LIN {X 0,Y 411.449,Z 252.234,A -85,B 0,C 180,E1 -10446.868,E2 -10446.868} C_VEL
LIN {X 0,Y 411.346,Z 252.246,A -85,B 0,C 180,E1 -10448.846,E2 -10448.846} C_VEL
LIN {X 0,Y 411.277,Z 252.254,A -85,B 0,C 180,E1 -10451.834,E2 -10451.834} C_VEL
LIN {X 0,Y 411.252,Z 252.259,A -85,B 0,C 180,E1 -10454.854,E2 -10454.854} C_VEL
LIN {X 0,Y 411.246,Z 252.261,A -85,B 0,C 180,E1 -10457.916,E2 -10457.916} C_VEL
LIN {X 0,Y 411.19,Z 252.268,A -85,B 0,C 180,E1 -10461.035,E2 -10461.035} C_VEL
LIN {X 0,Y 411.221,Z 252.266,A -85,B 0,C 180,E1 -10464.217,E2 -10464.217} C_VEL
LIN {X 0,Y 411.206,Z 252.269,A -85,B 0,C 180,E1 -10467.483,E2 -10467.483} C_VEL
LIN {X 0,Y 411.185,Z 252.27,A -85,B 0,C 180,E1 -10470.849,E2 -10470.849} C_VEL
LIN {X 0,Y 411.202,Z 252.265,A -85,B 0,C 180,E1 -10474.335,E2 -10474.335} C_VEL
LIN {X 0,Y 411.191,Z 252.266,A -85,B 0,C 180,E1 -10477.975,E2 -10477.975} C_VEL
LIN {X 0,Y 411.179,Z 252.263,A -85,B 0,C 180,E1 -10480.506,E2 -10480.506} C_VEL
LIN {X 0,Y 411.171,Z 252.27,A -85,B 0,C 180,E1 -10483.135,E2 -10483.135} C_VEL
LIN {X 0,Y 411.163,Z 252.271,A -85,B 0,C 180,E1 -10485.883,E2 -10485.883} C_VEL
LIN {X 0,Y 411.191,Z 252.402,A -85,B 0,C 180,E1 -10487.703,E2 -10487.703} C_VEL
LIN {X 0,Y 411.989,Z 257.108,A -85,B 0,C 180,E1 -10490.865,E2 -10490.865} C_VEL
LIN {X 0,Y 412.541,Z 261.129,A -85,B 0,C 180,E1 -10493.399,E2 -10493.399} C_VEL
LIN {X 0,Y 412.54,Z 265.204,A -85,B 0,C 180,E1 -10495.794,E2 -10495.794} C_VEL
LIN {X 0,Y 412.027,Z 271.404,A -85,B 0,C 180,E1 -10499.223,E2 -10499.223} C_VEL
LIN {X 0,Y 411.468,Z 277.887,A -85,B 0,C 180,E1 -10502.646,E2 -10502.646} C_VEL
LIN {X 0,Y 411.051,Z 285.054,A -85,B 0,C 180,E1 -10506.31,E2 -10506.31} C_VEL
LIN {X 0,Y 410.714,Z 291.422,A -85,B 0,C 180,E1 -10509.465,E2 -10509.465} C_VEL
LIN {X 0,Y 410.498,Z 296.726,A -85,B 0,C 180,E1 -10512.035,E2 -10512.035} C_VEL
LIN {X 0,Y 413.257,Z 309.763,A -85,B 0,C 180,E1 -10512.581,E2 -10512.581} C_VEL
LIN {X 0,Y 415.025,Z 322.416,A -85,B 0,C 180,E1 -10513.27,E2 -10513.27} C_VEL
LIN {X 0,Y 415.335,Z 326.719,A -85,B 0,C 180,E1 -10513.535,E2 -10513.535} C_VEL
LIN {X 0,Y 414.448,Z 339.122,A -85,B 0,C 180,E1 -10514.384,E2 -10514.384} C_VEL
LIN {X 0,Y 413.537,Z 350.197,A -85,B 0,C 180,E1 -10515.355,E2 -10515.355} C_VEL
LIN {X 0,Y 412.787,Z 360.22,A -85,B 0,C 180,E1 -10516.462,E2 -10516.462} C_VEL
LIN {X 0,Y 412.105,Z 369.286,A -85,B 0,C 180,E1 -10517.692,E2 -10517.692} C_VEL
LIN {X 0,Y 411.231,Z 378.148,A -85,B 0,C 180,E1 -10519.165,E2 -10519.165} C_VEL
LIN {X 0,Y 410.716,Z 385.289,A -85,B 0,C 180,E1 -10520.645,E2 -10520.645} C_VEL
LIN {X 0,Y 410.351,Z 391.005,A -85,B 0,C 180,E1 -10522.125,E2 -10522.125} C_VEL
LIN {X 0,Y 410.045,Z 395.958,A -85,B 0,C 180,E1 -10523.776,E2 -10523.776} C_VEL
LIN {X 0,Y 410.021,Z 398.967,A -85,B 0,C 180,E1 -10525.084,E2 -10525.084} C_VEL
LIN {X 0,Y 409.925,Z 402.002,A -85,B 0,C 180,E1 -10527.052,E2 -10527.052} C_VEL
LIN {X 0,Y 409.968,Z 402.928,A -85,B 0,C 180,E1 -10528.035,E2 -10528.035} C_VEL
LIN {X 0,Y 409.937,Z 403.449,A -85,B 0,C 180,E1 -10529.018,E2 -10529.018} C_VEL
LIN {X 0,Y 409.937,Z 403.25,A -85,B 0,C 180,E1 -10530.982,E2 -10530.982} C_VEL
LIN {X 0,Y 409.968,Z 402.571,A -85,B 0,C 180,E1 -10531.965,E2 -10531.965} C_VEL
LIN {X 0,Y 409.93,Z 401.489,A -85,B 0,C 180,E1 -10532.948,E2 -10532.948} C_VEL
LIN {X 0,Y 409.933,Z 399.952,A -85,B 0,C 180,E1 -10533.932,E2 -10533.932} C_VEL
LIN {X 0,Y 410.019,Z 396.857,A -85,B 0,C 180,E1 -10535.409,E2 -10535.409} C_VEL
LIN {X 0,Y 410.168,Z 392.694,A -85,B 0,C 180,E1 -10536.889,E2 -10536.889} C_VEL
LIN {X 0,Y 410.469,Z 386.328,A -85,B 0,C 180,E1 -10538.616,E2 -10538.616} C_VEL
LIN {X 0,Y 410.875,Z 379.388,A -85,B 0,C 180,E1 -10540.097,E2 -10540.097} C_VEL
LIN {X 0,Y 411.323,Z 372.293,A -85,B 0,C 180,E1 -10541.332,E2 -10541.332} C_VEL
LIN {X 0,Y 411.945,Z 363.724,A -85,B 0,C 180,E1 -10542.563,E2 -10542.563} C_VEL
LIN {X 0,Y 412.637,Z 353.121,A -85,B 0,C 180,E1 -10543.795,E2 -10543.795} C_VEL
LIN {X 0,Y 413.317,Z 342.609,A -85,B 0,C 180,E1 -10544.777,E2 -10544.777} C_VEL
LIN {X 0,Y 414.077,Z 331.039,A -85,B 0,C 180,E1 -10545.631,E2 -10545.631} C_VEL
LIN {X 0,Y 414.293,Z 324.137,A -85,B 0,C 180,E1 -10546.043,E2 -10546.043} C_VEL
LIN {X 0,Y 412.569,Z 311.085,A -85,B 0,C 180,E1 -10546.724,E2 -10546.724} C_VEL
LIN {X 0,Y 410.476,Z 298.087,A -85,B 0,C 180,E1 -10547.21,E2 -10547.21} C_VEL
LIN {X 0,Y 410.33,Z 296.882,A -85,B 0,C 180,E1 -10547.274,E2 -10547.274} C_VEL
LIN {X 0,Y 410.588,Z 289.945,A -85,B 0,C 180,E1 -10550.542,E2 -10550.542} C_VEL
LIN {X 0,Y 410.854,Z 283.341,A -85,B 0,C 180,E1 -10553.702,E2 -10553.702} C_VEL
LIN {X 0,Y 411.165,Z 277.823,A -85,B 0,C 180,E1 -10556.385,E2 -10556.385} C_VEL
LIN {X 0,Y 411.568,Z 271.207,A -85,B 0,C 180,E1 -10559.683,E2 -10559.683} C_VEL
LIN {X 0,Y 411.984,Z 264.559,A -85,B 0,C 180,E1 -10563.084,E2 -10563.084} C_VEL
LIN {X 0,Y 412.252,Z 260.131,A -85,B 0,C 180,E1 -10565.423,E2 -10565.423} C_VEL
LIN {X 0,Y 411.793,Z 255.662,A -85,B 0,C 180,E1 -10567.908,E2 -10567.908} C_VEL
LIN {X 0,Y 411.242,Z 252.261,A -85,B 0,C 180,E1 -10569.915,E2 -10569.915} C_VEL
LIN {X 0,Y 411.159,Z 252.27,A -85,B 0,C 180,E1 -10573.134,E2 -10573.134} C_VEL
LIN {X 0,Y 411.145,Z 252.268,A -85,B 0,C 180,E1 -10575.883,E2 -10575.883} C_VEL
LIN {X 0,Y 411.155,Z 252.268,A -85,B 0,C 180,E1 -10579.492,E2 -10579.492} C_VEL
LIN {X 0,Y 411.177,Z 252.265,A -85,B 0,C 180,E1 -10582.023,E2 -10582.023} C_VEL
LIN {X 0,Y 411.197,Z 252.264,A -85,B 0,C 180,E1 -10585.122,E2 -10585.122} C_VEL
LIN {X 0,Y 411.161,Z 252.268,A -85,B 0,C 180,E1 -10588.001,E2 -10588.001} C_VEL
LIN {X 0,Y 411.174,Z 252.266,A -85,B 0,C 180,E1 -10591.406,E2 -10591.406} C_VEL
LIN {X 0,Y 411.222,Z 252.261,A -85,B 0,C 180,E1 -10594.928,E2 -10594.928} C_VEL
LIN {X 0,Y 411.199,Z 252.265,A -85,B 0,C 180,E1 -10597.912,E2 -10597.912} C_VEL
LIN {X 0,Y 411.216,Z 252.261,A -85,B 0,C 180,E1 -10601.05,E2 -10601.05} C_VEL
LIN {X 0,Y 411.247,Z 252.26,A -85,B 0,C 180,E1 -10604.13,E2 -10604.13} C_VEL
LIN {X 0,Y 411.296,Z 252.251,A -85,B 0,C 180,E1 -10607.164,E2 -10607.164} C_VEL
LIN {X 0,Y 411.285,Z 252.254,A -85,B 0,C 180,E1 -10610.16,E2 -10610.16} C_VEL
LIN {X 0,Y 411.448,Z 252.232,A -85,B 0,C 180,E1 -10613.132,E2 -10613.132} C_VEL
LIN {X 0,Y 411.302,Z 252.25,A -85,B 0,C 180,E1 -10615.098,E2 -10615.098} C_VEL
LIN {X 0,Y 411.505,Z 252.227,A -85,B 0,C 180,E1 -10618.041,E2 -10618.041} C_VEL
LIN {X 0,Y 411.635,Z 252.211,A -85,B 0,C 180,E1 -10619.999,E2 -10619.999} C_VEL
LIN {X 0,Y 411.458,Z 252.231,A -85,B 0,C 180,E1 -10622.936,E2 -10622.936} C_VEL
LIN {X 0,Y 411.452,Z 252.232,A -85,B 0,C 180,E1 -10626.866,E2 -10626.866} C_VEL
LIN {X 0,Y 411.284,Z 252.255,A -85,B 0,C 180,E1 -10629.838,E2 -10629.838} C_VEL
LIN {X 0,Y 411.295,Z 252.252,A -85,B 0,C 180,E1 -10633.103,E2 -10633.103} C_VEL
LIN {X 0,Y 411.247,Z 252.258,A -85,B 0,C 180,E1 -10636.888,E2 -10636.888} C_VEL
LIN {X 0,Y 411.22,Z 252.261,A -85,B 0,C 180,E1 -10639.986,E2 -10639.986} C_VEL
LIN {X 0,Y 411.192,Z 252.265,A -85,B 0,C 180,E1 -10643.147,E2 -10643.147} C_VEL
LIN {X 0,Y 411.227,Z 252.259,A -85,B 0,C 180,E1 -10646.38,E2 -10646.38} C_VEL
LIN {X 0,Y 411.199,Z 252.264,A -85,B 0,C 180,E1 -10649.711,E2 -10649.711} C_VEL
LIN {X 0,Y 411.195,Z 252.268,A -85,B 0,C 180,E1 -10653.155,E2 -10653.155} C_VEL
LIN {X 0,Y 411.184,Z 252.265,A -85,B 0,C 180,E1 -10656.553,E2 -10656.553} C_VEL
LIN {X 0,Y 411.217,Z 252.259,A -85,B 0,C 180,E1 -10659.73,E2 -10659.73} C_VEL
LIN {X 0,Y 411.21,Z 252.263,A -85,B 0,C 180,E1 -10663.127,E2 -10663.127} C_VEL
LIN {X 0,Y 411.164,Z 252.265,A -85,B 0,C 180,E1 -10665.879,E2 -10665.879} C_VEL
LIN {X 0,Y 411.153,Z 252.273,A -85,B 0,C 180,E1 -10668.771,E2 -10668.771} C_VEL
LIN {X 0,Y 411.188,Z 252.263,A -85,B 0,C 180,E1 -10672.027,E2 -10672.027} C_VEL
LIN {X 0,Y 411.193,Z 252.262,A -85,B 0,C 180,E1 -10675.666,E2 -10675.666} C_VEL
LIN {X 0,Y 411.177,Z 252.265,A -85,B 0,C 180,E1 -10679.152,E2 -10679.152} C_VEL
LIN {X 0,Y 411.246,Z 252.259,A -85,B 0,C 180,E1 -10682.522,E2 -10682.522} C_VEL
LIN {X 0,Y 411.155,Z 252.269,A -85,B 0,C 180,E1 -10685.781,E2 -10685.781} C_VEL
LIN {X 0,Y 411.012,Z 252.288,A -85,B 0,C 180,E1 -10687.903,E2 -10687.903} C_VEL
LIN {X 0,Y 410.972,Z 253.172,A -85,B 0,C 180,E1 -10688.954,E2 -10688.954} C_VEL
LIN {X 0,Y 410.936,Z 255.861,A -85,B 0,C 180,E1 -10691.038,E2 -10691.038} C_VEL
LIN {X 0,Y 410.798,Z 259.931,A -85,B 0,C 180,E1 -10694.114,E2 -10694.114} C_VEL
LIN {X 0,Y 410.734,Z 264.145,A -85,B 0,C 180,E1 -10697.236,E2 -10697.236} C_VEL
LIN {X 0,Y 410.55,Z 269.533,A -85,B 0,C 180,E1 -10701.138,E2 -10701.138} C_VEL
LIN {X 0,Y 410.478,Z 273.682,A -85,B 0,C 180,E1 -10704.104,E2 -10704.104} C_VEL
LIN {X 0,Y 410.463,Z 276.293,A -85,B 0,C 180,E1 -10705.858,E2 -10705.858} C_VEL
LIN {X 0,Y 412.94,Z 289.606,A -85,B 0,C 180,E1 -10706.387,E2 -10706.387} C_VEL
LIN {X 0,Y 414.786,Z 300.337,A -85,B 0,C 180,E1 -10706.965,E2 -10706.965} C_VEL
LIN {X 0,Y 414.185,Z 312.098,A -85,B 0,C 180,E1 -10707.69,E2 -10707.69} C_VEL
LIN {X 0,Y 413.496,Z 322.814,A -85,B 0,C 180,E1 -10708.539,E2 -10708.539} C_VEL
LIN {X 0,Y 412.843,Z 333.725,A -85,B 0,C 180,E1 -10709.634,E2 -10709.634} C_VEL
LIN {X 0,Y 412.126,Z 342.64,A -85,B 0,C 180,E1 -10710.733,E2 -10710.733} C_VEL
LIN {X 0,Y 411.527,Z 350.815,A -85,B 0,C 180,E1 -10711.957,E2 -10711.957} C_VEL
LIN {X 0,Y 410.964,Z 358.837,A -85,B 0,C 180,E1 -10713.431,E2 -10713.431} C_VEL
LIN {X 0,Y 410.515,Z 365.289,A -85,B 0,C 180,E1 -10714.91,E2 -10714.91} C_VEL
LIN {X 0,Y 410.331,Z 371,A -85,B 0,C 180,E1 -10716.601,E2 -10716.601} C_VEL
LIN {X 0,Y 410.063,Z 375.459,A -85,B 0,C 180,E1 -10718.376,E2 -10718.376} C_VEL
LIN {X 0,Y 409.869,Z 378.544,A -85,B 0,C 180,E1 -10720.255,E2 -10720.255} C_VEL
LIN {X 0,Y 409.188,Z 379.493,A -85,B 0,C 180,E1 -10721.067,E2 -10721.067} C_VEL
LIN {X 0,Y 406.265,Z 380.427,A -85,B 0,C 180,E1 -10722.393,E2 -10722.393} C_VEL
LIN {X 0,Y 403.808,Z 380.668,A -85,B 0,C 180,E1 -10723.468,E2 -10723.468} C_VEL
LIN {X 0,Y 402.773,Z 380.524,A -85,B 0,C 180,E1 -10724.3,E2 -10724.3} C_VEL
LIN {X 0,Y 402.701,Z 380.36,A -85,B 0,C 180,E1 -10724.582,E2 -10724.582} C_VEL
LIN {X 0,Y 402.862,Z 378.906,A -85,B 0,C 180,E1 -10726.372,E2 -10726.372} C_VEL
LIN {X 0,Y 403.081,Z 375.863,A -85,B 0,C 180,E1 -10728.29,E2 -10728.29} C_VEL
LIN {X 0,Y 403.347,Z 372.347,A -85,B 0,C 180,E1 -10729.801,E2 -10729.801} C_VEL
LIN {X 0,Y 403.78,Z 367.273,A -85,B 0,C 180,E1 -10731.439,E2 -10731.439} C_VEL
LIN {X 0,Y 404.407,Z 360.409,A -85,B 0,C 180,E1 -10733.153,E2 -10733.153} C_VEL
LIN {X 0,Y 405.074,Z 353.084,A -85,B 0,C 180,E1 -10734.607,E2 -10734.607} C_VEL
LIN {X 0,Y 405.944,Z 344.026,A -85,B 0,C 180,E1 -10736.045,E2 -10736.045} C_VEL
LIN {X 0,Y 406.753,Z 334.707,A -85,B 0,C 180,E1 -10737.249,E2 -10737.249} C_VEL
LIN {X 0,Y 407.689,Z 324.192,A -85,B 0,C 180,E1 -10738.348,E2 -10738.348} C_VEL
LIN {X 0,Y 408.433,Z 313.724,A -85,B 0,C 180,E1 -10739.225,E2 -10739.225} C_VEL
LIN {X 0,Y 409.225,Z 302.753,A -85,B 0,C 180,E1 -10739.941,E2 -10739.941} C_VEL
LIN {X 0,Y 407.639,Z 293.422,A -85,B 0,C 180,E1 -10740.531,E2 -10740.531} C_VEL
LIN {X 0,Y 404.545,Z 281.297,A -85,B 0,C 180,E1 -10741.177,E2 -10741.177} C_VEL
LIN {X 0,Y 403.264,Z 276.621,A -85,B 0,C 180,E1 -10741.397,E2 -10741.397} C_VEL
LIN {X 0,Y 403.41,Z 273.295,A -85,B 0,C 180,E1 -10743.881,E2 -10743.881} C_VEL
LIN {X 0,Y 403.581,Z 268.536,A -85,B 0,C 180,E1 -10747.552,E2 -10747.552} C_VEL
LIN {X 0,Y 403.738,Z 265.304,A -85,B 0,C 180,E1 -10750.095,E2 -10750.095} C_VEL
LIN {X 0,Y 403.957,Z 261.659,A -85,B 0,C 180,E1 -10753.056,E2 -10753.056} C_VEL
LIN {X 0,Y 404.202,Z 258.197,A -85,B 0,C 180,E1 -10755.936,E2 -10755.936} C_VEL
LIN {X 0,Y 404.237,Z 255.081,A -85,B 0,C 180,E1 -10758.652,E2 -10758.652} C_VEL
LIN {X 0,Y 404.164,Z 253.629,A -85,B 0,C 180,E1 -10759.957,E2 -10759.957} C_VEL
LIN {X 0,Y 404.135,Z 253.148,A -85,B 0,C 180,E1 -10761.494,E2 -10761.494} C_VEL
LIN {X 0,Y 404.173,Z 253.143,A -85,B 0,C 180,E1 -10764.985,E2 -10764.985} C_VEL
LIN {X 0,Y 404.133,Z 253.148,A -85,B 0,C 180,E1 -10768.555,E2 -10768.555} C_VEL
LIN {X 0,Y 404.186,Z 253.14,A -85,B 0,C 180,E1 -10772.001,E2 -10772.001} C_VEL
LIN {X 0,Y 404.166,Z 253.141,A -85,B 0,C 180,E1 -10775.335,E2 -10775.335} C_VEL
LIN {X 0,Y 404.183,Z 253.138,A -85,B 0,C 180,E1 -10778.585,E2 -10778.585} C_VEL
LIN {X 0,Y 404.203,Z 253.135,A -85,B 0,C 180,E1 -10781.763,E2 -10781.763} C_VEL
LIN {X 0,Y 404.199,Z 253.136,A -85,B 0,C 180,E1 -10784.883,E2 -10784.883} C_VEL
LIN {X 0,Y 404.246,Z 253.131,A -85,B 0,C 180,E1 -10787.96,E2 -10787.96} C_VEL
LIN {X 0,Y 404.396,Z 253.111,A -85,B 0,C 180,E1 -10792.129,E2 -10792.129} C_VEL
LIN {X 0,Y 404.409,Z 253.109,A -85,B 0,C 180,E1 -10794.016,E2 -10794.016} C_VEL
LIN {X 0,Y 404.474,Z 253.102,A -85,B 0,C 180,E1 -10798.01,E2 -10798.01} C_VEL
LIN {X 0,Y 404.598,Z 253.085,A -85,B 0,C 180,E1 -10800.001,E2 -10800.001} C_VEL
LIN {X 0,Y 404.415,Z 253.11,A -85,B 0,C 180,E1 -10802.99,E2 -10802.99} C_VEL
LIN {X 0,Y 404.401,Z 253.111,A -85,B 0,C 180,E1 -10806.989,E2 -10806.989} C_VEL
LIN {X 0,Y 404.251,Z 253.13,A -85,B 0,C 180,E1 -10810.013,E2 -10810.013} C_VEL
LIN {X 0,Y 404.26,Z 253.129,A -85,B 0,C 180,E1 -10813.213,E2 -10813.213} C_VEL
LIN {X 0,Y 404.21,Z 253.139,A -85,B 0,C 180,E1 -10817.008,E2 -10817.008} C_VEL
LIN {X 0,Y 404.158,Z 253.146,A -85,B 0,C 180,E1 -10820.353,E2 -10820.353} C_VEL
LIN {X 0,Y 404.164,Z 253.145,A -85,B 0,C 180,E1 -10823.576,E2 -10823.576} C_VEL
LIN {X 0,Y 404.168,Z 253.145,A -85,B 0,C 180,E1 -10825.769,E2 -10825.769} C_VEL
LIN {X 0,Y 404.155,Z 253.147,A -85,B 0,C 180,E1 -10829.138,E2 -10829.138} C_VEL
LIN {X 0,Y 404.137,Z 253.146,A -85,B 0,C 180,E1 -10832.623,E2 -10832.623} C_VEL
LIN {X 0,Y 404.177,Z 253.141,A -85,B 0,C 180,E1 -10835.191,E2 -10835.191} C_VEL
LIN {X 0,Y 404.152,Z 253.142,A -85,B 0,C 180,E1 -10838.758,E2 -10838.758} C_VEL
LIN {X 0,Y 404.121,Z 253.146,A -85,B 0,C 180,E1 -10841.601,E2 -10841.601} C_VEL
LIN {X 0,Y 404.144,Z 253.136,A -85,B 0,C 180,E1 -10844.523,E2 -10844.523} C_VEL
LIN {X 0,Y 404.148,Z 253.242,A -85,B 0,C 180,E1 -10847.298,E2 -10847.298} C_VEL
LIN {X 0,Y 404.833,Z 257.174,A -85,B 0,C 180,E1 -10850.035,E2 -10850.035} C_VEL
LIN {X 0,Y 405.473,Z 261.538,A -85,B 0,C 180,E1 -10852.875,E2 -10852.875} C_VEL
LIN {X 0,Y 405.591,Z 265.254,A -85,B 0,C 180,E1 -10855.124,E2 -10855.124} C_VEL
LIN {X 0,Y 405.26,Z 269.341,A -85,B 0,C 180,E1 -10857.48,E2 -10857.48} C_VEL
LIN {X 0,Y 404.841,Z 274.314,A -85,B 0,C 180,E1 -10860.228,E2 -10860.228} C_VEL
LIN {X 0,Y 404.279,Z 280.794,A -85,B 0,C 180,E1 -10863.687,E2 -10863.687} C_VEL
LIN {X 0,Y 403.902,Z 287.706,A -85,B 0,C 180,E1 -10867.254,E2 -10867.254} C_VEL
LIN {X 0,Y 403.56,Z 293.416,A -85,B 0,C 180,E1 -10870.123,E2 -10870.123} C_VEL
LIN {X 0,Y 403.447,Z 296.645,A -85,B 0,C 180,E1 -10871.655,E2 -10871.655} C_VEL
LIN {X 0,Y 406.328,Z 309.623,A -85,B 0,C 180,E1 -10872.223,E2 -10872.223} C_VEL
LIN {X 0,Y 408.108,Z 321.885,A -85,B 0,C 180,E1 -10872.909,E2 -10872.909} C_VEL
LIN {X 0,Y 408.572,Z 327.244,A -85,B 0,C 180,E1 -10873.255,E2 -10873.255} C_VEL
LIN {X 0,Y 407.646,Z 339.5,A -85,B 0,C 180,E1 -10874.116,E2 -10874.116} C_VEL
LIN {X 0,Y 406.684,Z 350.557,A -85,B 0,C 180,E1 -10875.113,E2 -10875.113} C_VEL
LIN {X 0,Y 405.889,Z 360.376,A -85,B 0,C 180,E1 -10876.227,E2 -10876.227} C_VEL
LIN {X 0,Y 405.16,Z 369.383,A -85,B 0,C 180,E1 -10877.478,E2 -10877.478} C_VEL
LIN {X 0,Y 404.228,Z 378.195,A -85,B 0,C 180,E1 -10878.975,E2 -10878.975} C_VEL
LIN {X 0,Y 403.684,Z 385.28,A -85,B 0,C 180,E1 -10880.48,E2 -10880.48} C_VEL
LIN {X 0,Y 403.296,Z 390.949,A -85,B 0,C 180,E1 -10881.986,E2 -10881.986} C_VEL
LIN {X 0,Y 402.942,Z 396.246,A -85,B 0,C 180,E1 -10883.82,E2 -10883.82} C_VEL
LIN {X 0,Y 402.933,Z 398.844,A -85,B 0,C 180,E1 -10884.997,E2 -10884.997} C_VEL
LIN {X 0,Y 402.824,Z 401.848,A -85,B 0,C 180,E1 -10887,E2 -10887} C_VEL
LIN {X 0,Y 402.866,Z 402.76,A -85,B 0,C 180,E1 -10888.001,E2 -10888.001} C_VEL
LIN {X 0,Y 402.864,Z 403.257,A -85,B 0,C 180,E1 -10889,E2 -10889} C_VEL
LIN {X 0,Y 402.864,Z 403.031,A -85,B 0,C 180,E1 -10891,E2 -10891} C_VEL
LIN {X 0,Y 402.881,Z 402.339,A -85,B 0,C 180,E1 -10891.999,E2 -10891.999} C_VEL
LIN {X 0,Y 402.829,Z 401.232,A -85,B 0,C 180,E1 -10893,E2 -10893} C_VEL
LIN {X 0,Y 402.854,Z 399.679,A -85,B 0,C 180,E1 -10894.001,E2 -10894.001} C_VEL
LIN {X 0,Y 402.917,Z 396.553,A -85,B 0,C 180,E1 -10895.505,E2 -10895.505} C_VEL
LIN {X 0,Y 403.08,Z 392.356,A -85,B 0,C 180,E1 -10897.01,E2 -10897.01} C_VEL
LIN {X 0,Y 403.406,Z 385.953,A -85,B 0,C 180,E1 -10898.768,E2 -10898.768} C_VEL
LIN {X 0,Y 403.816,Z 378.963,A -85,B 0,C 180,E1 -10900.276,E2 -10900.276} C_VEL
LIN {X 0,Y 404.447,Z 370.19,A -85,B 0,C 180,E1 -10901.781,E2 -10901.781} C_VEL
LIN {X 0,Y 405.07,Z 361.192,A -85,B 0,C 180,E1 -10903.035,E2 -10903.035} C_VEL
LIN {X 0,Y 405.756,Z 351.295,A -85,B 0,C 180,E1 -10904.161,E2 -10904.161} C_VEL
LIN {X 0,Y 406.523,Z 340.37,A -85,B 0,C 180,E1 -10905.158,E2 -10905.158} C_VEL
LIN {X 0,Y 407.314,Z 328.101,A -85,B 0,C 180,E1 -10906.026,E2 -10906.026} C_VEL
LIN {X 0,Y 407.049,Z 322.118,A -85,B 0,C 180,E1 -10906.388,E2 -10906.388} C_VEL
LIN {X 0,Y 405.243,Z 309.092,A -85,B 0,C 180,E1 -10907.056,E2 -10907.056} C_VEL
LIN {X 0,Y 403.259,Z 296.712,A -85,B 0,C 180,E1 -10907.528,E2 -10907.528} C_VEL
LIN {X 0,Y 403.549,Z 289.665,A -85,B 0,C 180,E1 -10910.917,E2 -10910.917} C_VEL
LIN {X 0,Y 403.853,Z 283.072,A -85,B 0,C 180,E1 -10914.139,E2 -10914.139} C_VEL
LIN {X 0,Y 404.131,Z 277.567,A -85,B 0,C 180,E1 -10916.881,E2 -10916.881} C_VEL
LIN {X 0,Y 404.59,Z 270.943,A -85,B 0,C 180,E1 -10920.248,E2 -10920.248} C_VEL
LIN {X 0,Y 405.02,Z 264.295,A -85,B 0,C 180,E1 -10923.729,E2 -10923.729} C_VEL
LIN {X 0,Y 405.16,Z 259.864,A -85,B 0,C 180,E1 -10926.14,E2 -10926.14} C_VEL
LIN {X 0,Y 404.568,Z 255.407,A -85,B 0,C 180,E1 -10928.709,E2 -10928.709} C_VEL
LIN {X 0,Y 404.199,Z 253.139,A -85,B 0,C 180,E1 -10930.088,E2 -10930.088} C_VEL
LIN {X 0,Y 404.116,Z 253.144,A -85,B 0,C 180,E1 -10934.077,E2 -10934.077} C_VEL
LIN {X 0,Y 404.073,Z 253.151,A -85,B 0,C 180,E1 -10937.286,E2 -10937.286} C_VEL
LIN {X 0,Y 404.13,Z 253.142,A -85,B 0,C 180,E1 -10939.95,E2 -10939.95} C_VEL
LIN {X 0,Y 404.127,Z 253.145,A -85,B 0,C 180,E1 -10943.125,E2 -10943.125} C_VEL
LIN {X 0,Y 404.134,Z 253.144,A -85,B 0,C 180,E1 -10946.186,E2 -10946.186} C_VEL
LIN {X 0,Y 404.14,Z 253.142,A -85,B 0,C 180,E1 -10949.713,E2 -10949.713} C_VEL
LIN {X 0,Y 404.119,Z 253.146,A -85,B 0,C 180,E1 -10953.116,E2 -10953.116} C_VEL
LIN {X 0,Y 404.152,Z 253.143,A -85,B 0,C 180,E1 -10956.423,E2 -10956.423} C_VEL
LIN {X 0,Y 404.186,Z 253.138,A -85,B 0,C 180,E1 -10959.873,E2 -10959.873} C_VEL
LIN {X 0,Y 404.21,Z 253.134,A -85,B 0,C 180,E1 -10962.992,E2 -10962.992} C_VEL
LIN {X 0,Y 404.276,Z 253.126,A -85,B 0,C 180,E1 -10966.938,E2 -10966.938} C_VEL
LIN {X 0,Y 404.251,Z 253.131,A -85,B 0,C 180,E1 -10969.987,E2 -10969.987} C_VEL
LIN {X 0,Y 404.395,Z 253.11,A -85,B 0,C 180,E1 -10973.011,E2 -10973.011} C_VEL
LIN {X 0,Y 404.274,Z 253.126,A -85,B 0,C 180,E1 -10975.012,E2 -10975.012} C_VEL
LIN {X 0,Y 404.474,Z 253.103,A -85,B 0,C 180,E1 -10978.007,E2 -10978.007} C_VEL
LIN {X 0,Y 404.604,Z 253.087,A -85,B 0,C 180,E1 -10979.999,E2 -10979.999} C_VEL
LIN {X 0,Y 404.415,Z 253.108,A -85,B 0,C 180,E1 -10982.987,E2 -10982.987} C_VEL
LIN {X 0,Y 404.403,Z 253.11,A -85,B 0,C 180,E1 -10986.986,E2 -10986.986} C_VEL
LIN {X 0,Y 404.25,Z 253.131,A -85,B 0,C 180,E1 -10990.011,E2 -10990.011} C_VEL
LIN {X 0,Y 404.256,Z 253.129,A -85,B 0,C 180,E1 -10993.21,E2 -10993.21} C_VEL
LIN {X 0,Y 404.205,Z 253.135,A -85,B 0,C 180,E1 -10997.006,E2 -10997.006} C_VEL
LIN {X 0,Y 404.153,Z 253.14,A -85,B 0,C 180,E1 -11000.351,E2 -11000.351} C_VEL
LIN {X 0,Y 404.158,Z 253.143,A -85,B 0,C 180,E1 -11003.574,E2 -11003.574} C_VEL
LIN {X 0,Y 404.172,Z 253.139,A -85,B 0,C 180,E1 -11005.766,E2 -11005.766} C_VEL
LIN {X 0,Y 404.186,Z 253.136,A -85,B 0,C 180,E1 -11007.999,E2 -11007.999} C_VEL
LIN {X 0,Y 404.131,Z 253.145,A -85,B 0,C 180,E1 -11011.558,E2 -11011.558} C_VEL
LIN {X 0,Y 404.174,Z 253.141,A -85,B 0,C 180,E1 -11015.015,E2 -11015.015} C_VEL
LIN {X 0,Y 404.152,Z 253.142,A -85,B 0,C 180,E1 -11018.755,E2 -11018.755} C_VEL
LIN {X 0,Y 404.179,Z 253.136,A -85,B 0,C 180,E1 -11021.61,E2 -11021.61} C_VEL
LIN {X 0,Y 404.178,Z 253.138,A -85,B 0,C 180,E1 -11024.528,E2 -11024.528} C_VEL
LIN {X 0,Y 404.127,Z 253.143,A -85,B 0,C 180,E1 -11027.296,E2 -11027.296} C_VEL
LIN {X 0,Y 404.157,Z 253.138,A -85,B 0,C 180,E1 -11029.955,E2 -11029.955} C_VEL
LIN {X 0,Y 404.127,Z 253.144,A -85,B 0,C 180,E1 -11033.124,E2 -11033.124} C_VEL
LIN {X 0,Y 404.133,Z 253.144,A -85,B 0,C 180,E1 -11036.187,E2 -11036.187} C_VEL
LIN {X 0,Y 404.133,Z 253.142,A -85,B 0,C 180,E1 -11039.715,E2 -11039.715} C_VEL
LIN {X 0,Y 404.18,Z 253.137,A -85,B 0,C 180,E1 -11043.122,E2 -11043.122} C_VEL
LIN {X 0,Y 404.07,Z 253.153,A -85,B 0,C 180,E1 -11046.42,E2 -11046.42} C_VEL
LIN {X 0,Y 404.033,Z 253.155,A -85,B 0,C 180,E1 -11047.501,E2 -11047.501} C_VEL
LIN {X 0,Y 403.911,Z 253.541,A -85,B 0,C 180,E1 -11048.568,E2 -11048.568} C_VEL
LIN {X 0,Y 403.921,Z 256.251,A -85,B 0,C 180,E1 -11050.696,E2 -11050.696} C_VEL
LIN {X 0,Y 403.777,Z 260.321,A -85,B 0,C 180,E1 -11053.83,E2 -11053.83} C_VEL
LIN {X 0,Y 403.678,Z 264.724,A -85,B 0,C 180,E1 -11057.142,E2 -11057.142} C_VEL
LIN {X 0,Y 403.471,Z 269.943,A -85,B 0,C 180,E1 -11060.981,E2 -11060.981} C_VEL
LIN {X 0,Y 403.426,Z 274.141,A -85,B 0,C 180,E1 -11064,E2 -11064} C_VEL
LIN {X 0,Y 403.422,Z 276.478,A -85,B 0,C 180,E1 -11065.598,E2 -11065.598} C_VEL
LIN {X 0,Y 405.857,Z 289.453,A -85,B 0,C 180,E1 -11066.121,E2 -11066.121} C_VEL
LIN {X 0,Y 407.861,Z 300.461,A -85,B 0,C 180,E1 -11066.728,E2 -11066.728} C_VEL
LIN {X 0,Y 407.228,Z 313.099,A -85,B 0,C 180,E1 -11067.527,E2 -11067.527} C_VEL
LIN {X 0,Y 406.453,Z 324.935,A -85,B 0,C 180,E1 -11068.514,E2 -11068.514} C_VEL
LIN {X 0,Y 405.74,Z 335.48,A -85,B 0,C 180,E1 -11069.628,E2 -11069.628} C_VEL
LIN {X 0,Y 405.054,Z 344.128,A -85,B 0,C 180,E1 -11070.746,E2 -11070.746} C_VEL
LIN {X 0,Y 404.417,Z 352.096,A -85,B 0,C 180,E1 -11071.992,E2 -11071.992} C_VEL
LIN {X 0,Y 403.884,Z 359.905,A -85,B 0,C 180,E1 -11073.492,E2 -11073.492} C_VEL
LIN {X 0,Y 403.42,Z 366.158,A -85,B 0,C 180,E1 -11074.997,E2 -11074.997} C_VEL
LIN {X 0,Y 403.243,Z 371.346,A -85,B 0,C 180,E1 -11076.584,E2 -11076.584} C_VEL
LIN {X 0,Y 403.029,Z 374.978,A -85,B 0,C 180,E1 -11078.019,E2 -11078.019} C_VEL
LIN {X 0,Y 402.861,Z 376.972,A -85,B 0,C 180,E1 -11079.033,E2 -11079.033} C_VEL
LIN {X 0,Y 402.772,Z 378.764,A -85,B 0,C 180,E1 -11080.246,E2 -11080.246} C_VEL
LIN {X 0,Y 402.801,Z 380.368,A -85,B 0,C 180,E1 -11082.085,E2 -11082.085} C_VEL
LIN {X 0,Y 402.701,Z 380.682,A -85,B 0,C 180,E1 -11083.113,E2 -11083.113} C_VEL
LIN {X 0,Y 402.701,Z 380.36,A -85,B 0,C 180,E1 -11084.582,E2 -11084.582} C_VEL
LIN {X 0,Y 402.082,Z 379.899,A -85,B 0,C 180,E1 -11085.414,E2 -11085.414} C_VEL
LIN {X 0,Y 399.332,Z 378.588,A -85,B 0,C 180,E1 -11086.764,E2 -11086.764} C_VEL
LIN {X 0,Y 397.047,Z 377.068,A -85,B 0,C 180,E1 -11087.842,E2 -11087.842} C_VEL
LIN {X 0,Y 396.141,Z 375.586,A -85,B 0,C 180,E1 -11088.662,E2 -11088.662} C_VEL
LIN {X 0,Y 396.109,Z 375.007,A -85,B 0,C 180,E1 -11088.937,E2 -11088.937} C_VEL
LIN {X 0,Y 396.521,Z 370.309,A -85,B 0,C 180,E1 -11090.761,E2 -11090.761} C_VEL
LIN {X 0,Y 397.126,Z 363.752,A -85,B 0,C 180,E1 -11092.638,E2 -11092.638} C_VEL
LIN {X 0,Y 397.812,Z 356.506,A -85,B 0,C 180,E1 -11094.251,E2 -11094.251} C_VEL
LIN {X 0,Y 398.693,Z 348.09,A -85,B 0,C 180,E1 -11095.737,E2 -11095.737} C_VEL
LIN {X 0,Y 399.589,Z 338.796,A -85,B 0,C 180,E1 -11097.07,E2 -11097.07} C_VEL
LIN {X 0,Y 400.574,Z 328.368,A -85,B 0,C 180,E1 -11098.275,E2 -11098.275} C_VEL
LIN {X 0,Y 401.527,Z 316.589,A -85,B 0,C 180,E1 -11099.346,E2 -11099.346} C_VEL
LIN {X 0,Y 402.454,Z 304.784,A -85,B 0,C 180,E1 -11100.174,E2 -11100.174} C_VEL
LIN {X 0,Y 401.863,Z 299.29,A -85,B 0,C 180,E1 -11100.539,E2 -11100.539} C_VEL
LIN {X 0,Y 399.046,Z 286.807,A -85,B 0,C 180,E1 -11101.291,E2 -11101.291} C_VEL
LIN {X 0,Y 396.217,Z 276.808,A -85,B 0,C 180,E1 -11101.809,E2 -11101.809} C_VEL
LIN {X 0,Y 396.381,Z 273.194,A -85,B 0,C 180,E1 -11104.566,E2 -11104.566} C_VEL
LIN {X 0,Y 396.6,Z 268.402,A -85,B 0,C 180,E1 -11108.331,E2 -11108.331} C_VEL
LIN {X 0,Y 396.812,Z 263.973,A -85,B 0,C 180,E1 -11111.94,E2 -11111.94} C_VEL
LIN {X 0,Y 397.09,Z 260.236,A -85,B 0,C 180,E1 -11115.067,E2 -11115.067} C_VEL
LIN {X 0,Y 397.235,Z 256.878,A -85,B 0,C 180,E1 -11117.993,E2 -11117.993} C_VEL
LIN {X 0,Y 397.086,Z 254.22,A -85,B 0,C 180,E1 -11120.422,E2 -11120.422} C_VEL
LIN {X 0,Y 397.088,Z 254.023,A -85,B 0,C 180,E1 -11123.006,E2 -11123.006} C_VEL
LIN {X 0,Y 397.106,Z 254.024,A -85,B 0,C 180,E1 -11126.283,E2 -11126.283} C_VEL
LIN {X 0,Y 397.102,Z 254.023,A -85,B 0,C 180,E1 -11130.134,E2 -11130.134} C_VEL
LIN {X 0,Y 397.183,Z 254.01,A -85,B 0,C 180,E1 -11132.611,E2 -11132.611} C_VEL
LIN {X 0,Y 397.123,Z 254.019,A -85,B 0,C 180,E1 -11135.983,E2 -11135.983} C_VEL
LIN {X 0,Y 397.144,Z 254.015,A -85,B 0,C 180,E1 -11139.274,E2 -11139.274} C_VEL
LIN {X 0,Y 397.173,Z 254.011,A -85,B 0,C 180,E1 -11142.845,E2 -11142.845} C_VEL
LIN {X 0,Y 397.167,Z 254.01,A -85,B 0,C 180,E1 -11145.658,E2 -11145.658} C_VEL
LIN {X 0,Y 397.189,Z 254.011,A -85,B 0,C 180,E1 -11148.778,E2 -11148.778} C_VEL
LIN {X 0,Y 397.352,Z 253.989,A -85,B 0,C 180,E1 -11152.076,E2 -11152.076} C_VEL
LIN {X 0,Y 397.244,Z 254.003,A -85,B 0,C 180,E1 -11154.926,E2 -11154.926} C_VEL
LIN {X 0,Y 397.443,Z 253.978,A -85,B 0,C 180,E1 -11157.974,E2 -11157.974} C_VEL
LIN {X 0,Y 397.568,Z 253.961,A -85,B 0,C 180,E1 -11160.001,E2 -11160.001} C_VEL
LIN {X 0,Y 397.373,Z 253.987,A -85,B 0,C 180,E1 -11163.043,E2 -11163.043} C_VEL
LIN {X 0,Y 397.354,Z 253.989,A -85,B 0,C 180,E1 -11167.113,E2 -11167.113} C_VEL
LIN {X 0,Y 397.211,Z 254.007,A -85,B 0,C 180,E1 -11170.192,E2 -11170.192} C_VEL
LIN {X 0,Y 397.22,Z 254.005,A -85,B 0,C 180,E1 -11173.322,E2 -11173.322} C_VEL
LIN {X 0,Y 397.176,Z 254.015,A -85,B 0,C 180,E1 -11177.156,E2 -11177.156} C_VEL
LIN {X 0,Y 397.097,Z 254.023,A -85,B 0,C 180,E1 -11180.731,E2 -11180.731} C_VEL
LIN {X 0,Y 397.127,Z 254.021,A -85,B 0,C 180,E1 -11184.02,E2 -11184.02} C_VEL
LIN {X 0,Y 397.136,Z 254.022,A -85,B 0,C 180,E1 -11187.396,E2 -11187.396} C_VEL
LIN {X 0,Y 397.074,Z 254.028,A -85,B 0,C 180,E1 -11190.884,E2 -11190.884} C_VEL
LIN {X 0,Y 397.122,Z 254.019,A -85,B 0,C 180,E1 -11194.495,E2 -11194.495} C_VEL
LIN {X 0,Y 397.1,Z 254.023,A -85,B 0,C 180,E1 -11198.276,E2 -11198.276} C_VEL
LIN {X 0,Y 397.087,Z 254.02,A -85,B 0,C 180,E1 -11200.91,E2 -11200.91} C_VEL
LIN {X 0,Y 397.1,Z 254.022,A -85,B 0,C 180,E1 -11203.65,E2 -11203.65} C_VEL
LIN {X 0,Y 397.1,Z 254.074,A -85,B 0,C 180,E1 -11206.876,E2 -11206.876} C_VEL
LIN {X 0,Y 397.713,Z 257.682,A -85,B 0,C 180,E1 -11209.453,E2 -11209.453} C_VEL
LIN {X 0,Y 398.425,Z 262.288,A -85,B 0,C 180,E1 -11212.541,E2 -11212.541} C_VEL
LIN {X 0,Y 398.587,Z 266.299,A -85,B 0,C 180,E1 -11215.038,E2 -11215.038} C_VEL
LIN {X 0,Y 398.152,Z 271.416,A -85,B 0,C 180,E1 -11218.026,E2 -11218.026} C_VEL
LIN {X 0,Y 397.67,Z 276.605,A -85,B 0,C 180,E1 -11220.922,E2 -11220.922} C_VEL
LIN {X 0,Y 397.111,Z 283.913,A -85,B 0,C 180,E1 -11224.866,E2 -11224.866} C_VEL
LIN {X 0,Y 396.733,Z 290.229,A -85,B 0,C 180,E1 -11228.161,E2 -11228.161} C_VEL
LIN {X 0,Y 396.398,Z 296.384,A -85,B 0,C 180,E1 -11231.256,E2 -11231.256} C_VEL
LIN {X 0,Y 399.45,Z 309.853,A -85,B 0,C 180,E1 -11231.868,E2 -11231.868} C_VEL
LIN {X 0,Y 401.299,Z 322.142,A -85,B 0,C 180,E1 -11232.581,E2 -11232.581} C_VEL
LIN {X 0,Y 401.698,Z 329.828,A -85,B 0,C 180,E1 -11233.091,E2 -11233.091} C_VEL
LIN {X 0,Y 400.716,Z 341.427,A -85,B 0,C 180,E1 -11233.965,E2 -11233.965} C_VEL
LIN {X 0,Y 399.611,Z 353.087,A -85,B 0,C 180,E1 -11235.096,E2 -11235.096} C_VEL
LIN {X 0,Y 398.839,Z 362.493,A -85,B 0,C 180,E1 -11236.239,E2 -11236.239} C_VEL
LIN {X 0,Y 398.066,Z 371.109,A -85,B 0,C 180,E1 -11237.51,E2 -11237.51} C_VEL
LIN {X 0,Y 397.145,Z 379.501,A -85,B 0,C 180,E1 -11239.034,E2 -11239.034} C_VEL
LIN {X 0,Y 396.576,Z 386.274,A -85,B 0,C 180,E1 -11240.565,E2 -11240.565} C_VEL
LIN {X 0,Y 396.154,Z 392.514,A -85,B 0,C 180,E1 -11242.354,E2 -11242.354} C_VEL
LIN {X 0,Y 395.831,Z 397.271,A -85,B 0,C 180,E1 -11244.194,E2 -11244.194} C_VEL
LIN {X 0,Y 395.776,Z 400.411,A -85,B 0,C 180,E1 -11245.927,E2 -11245.927} C_VEL
LIN {X 0,Y 395.763,Z 402.596,A -85,B 0,C 180,E1 -11247.965,E2 -11247.965} C_VEL
LIN {X 0,Y 395.792,Z 403.065,A -85,B 0,C 180,E1 -11248.983,E2 -11248.983} C_VEL
LIN {X 0,Y 395.793,Z 402.809,A -85,B 0,C 180,E1 -11251.017,E2 -11251.017} C_VEL
LIN {X 0,Y 395.779,Z 402.102,A -85,B 0,C 180,E1 -11252.035,E2 -11252.035} C_VEL
LIN {X 0,Y 395.732,Z 400.964,A -85,B 0,C 180,E1 -11253.054,E2 -11253.054} C_VEL
LIN {X 0,Y 395.777,Z 399.396,A -85,B 0,C 180,E1 -11254.073,E2 -11254.073} C_VEL
LIN {X 0,Y 395.829,Z 395.746,A -85,B 0,C 180,E1 -11255.804,E2 -11255.804} C_VEL
LIN {X 0,Y 396.068,Z 390.362,A -85,B 0,C 180,E1 -11257.648,E2 -11257.648} C_VEL
LIN {X 0,Y 396.477,Z 383.367,A -85,B 0,C 180,E1 -11259.437,E2 -11259.437} C_VEL
LIN {X 0,Y 396.964,Z 375.786,A -85,B 0,C 180,E1 -11260.971,E2 -11260.971} C_VEL
LIN {X 0,Y 397.627,Z 368.046,A -85,B 0,C 180,E1 -11262.245,E2 -11262.245} C_VEL
LIN {X 0,Y 398.279,Z 359.07,A -85,B 0,C 180,E1 -11263.463,E2 -11263.463} C_VEL
LIN {X 0,Y 398.999,Z 348.074,A -85,B 0,C 180,E1 -11264.667,E2 -11264.667} C_VEL
LIN {X 0,Y 399.847,Z 336.393,A -85,B 0,C 180,E1 -11265.678,E2 -11265.678} C_VEL
LIN {X 0,Y 400.436,Z 325.959,A -85,B 0,C 180,E1 -11266.386,E2 -11266.386} C_VEL
LIN {X 0,Y 398.763,Z 312.947,A -85,B 0,C 180,E1 -11267.124,E2 -11267.124} C_VEL
LIN {X 0,Y 396.635,Z 299.439,A -85,B 0,C 180,E1 -11267.679,E2 -11267.679} C_VEL
LIN {X 0,Y 396.19,Z 296.549,A -85,B 0,C 180,E1 -11267.784,E2 -11267.784} C_VEL
LIN {X 0,Y 396.526,Z 289.37,A -85,B 0,C 180,E1 -11271.305,E2 -11271.305} C_VEL
LIN {X 0,Y 396.892,Z 281.692,A -85,B 0,C 180,E1 -11275.149,E2 -11275.149} C_VEL
LIN {X 0,Y 397.291,Z 275.075,A -85,B 0,C 180,E1 -11278.53,E2 -11278.53} C_VEL
LIN {X 0,Y 397.682,Z 269.583,A -85,B 0,C 180,E1 -11281.414,E2 -11281.414} C_VEL
LIN {X 0,Y 398.173,Z 262.927,A -85,B 0,C 180,E1 -11285.004,E2 -11285.004} C_VEL
LIN {X 0,Y 397.921,Z 258.793,A -85,B 0,C 180,E1 -11287.364,E2 -11287.364} C_VEL
LIN {X 0,Y 397.152,Z 254.017,A -85,B 0,C 180,E1 -11290.227,E2 -11290.227} C_VEL
LIN {X 0,Y 397.084,Z 254.02,A -85,B 0,C 180,E1 -11293.65,E2 -11293.65} C_VEL
LIN {X 0,Y 397.033,Z 254.029,A -85,B 0,C 180,E1 -11296.53,E2 -11296.53} C_VEL
LIN {X 0,Y 397.083,Z 254.023,A -85,B 0,C 180,E1 -11300.418,E2 -11300.418} C_VEL
LIN {X 0,Y 397.089,Z 254.022,A -85,B 0,C 180,E1 -11303.003,E2 -11303.003} C_VEL
LIN {X 0,Y 397.108,Z 254.021,A -85,B 0,C 180,E1 -11306.725,E2 -11306.725} C_VEL
LIN {X 0,Y 397.113,Z 254.02,A -85,B 0,C 180,E1 -11310.294,E2 -11310.294} C_VEL
LIN {X 0,Y 397.083,Z 254.021,A -85,B 0,C 180,E1 -11313.737,E2 -11313.737} C_VEL
LIN {X 0,Y 397.098,Z 254.02,A -85,B 0,C 180,E1 -11317.084,E2 -11317.084} C_VEL
LIN {X 0,Y 397.142,Z 254.017,A -85,B 0,C 180,E1 -11320.351,E2 -11320.351} C_VEL
LIN {X 0,Y 397.16,Z 254.012,A -85,B 0,C 180,E1 -11323.552,E2 -11323.552} C_VEL
LIN {X 0,Y 397.223,Z 254.005,A -85,B 0,C 180,E1 -11326.701,E2 -11326.701} C_VEL
LIN {X 0,Y 397.21,Z 254.008,A -85,B 0,C 180,E1 -11329.808,E2 -11329.808} C_VEL
LIN {X 0,Y 397.345,Z 253.989,A -85,B 0,C 180,E1 -11332.887,E2 -11332.887} C_VEL
LIN {X 0,Y 397.246,Z 254.001,A -85,B 0,C 180,E1 -11334.924,E2 -11334.924} C_VEL
LIN {X 0,Y 397.443,Z 253.979,A -85,B 0,C 180,E1 -11337.972,E2 -11337.972} C_VEL
LIN {X 0,Y 397.574,Z 253.963,A -85,B 0,C 180,E1 -11339.999,E2 -11339.999} C_VEL
LIN {X 0,Y 397.374,Z 253.985,A -85,B 0,C 180,E1 -11343.04,E2 -11343.04} C_VEL
LIN {X 0,Y 397.355,Z 253.988,A -85,B 0,C 180,E1 -11347.111,E2 -11347.111} C_VEL
LIN {X 0,Y 397.209,Z 254.007,A -85,B 0,C 180,E1 -11350.19,E2 -11350.19} C_VEL
LIN {X 0,Y 397.217,Z 254.006,A -85,B 0,C 180,E1 -11353.32,E2 -11353.32} C_VEL
LIN {X 0,Y 397.171,Z 254.012,A -85,B 0,C 180,E1 -11357.154,E2 -11357.154} C_VEL
LIN {X 0,Y 397.092,Z 254.02,A -85,B 0,C 180,E1 -11360.729,E2 -11360.729} C_VEL
LIN {X 0,Y 397.122,Z 254.016,A -85,B 0,C 180,E1 -11364.017,E2 -11364.017} C_VEL
LIN {X 0,Y 397.183,Z 254.013,A -85,B 0,C 180,E1 -11367.389,E2 -11367.389} C_VEL
LIN {X 0,Y 397.073,Z 254.024,A -85,B 0,C 180,E1 -11370.881,E2 -11370.881} C_VEL
LIN {X 0,Y 397.114,Z 254.017,A -85,B 0,C 180,E1 -11374.493,E2 -11374.493} C_VEL
LIN {X 0,Y 397.098,Z 254.018,A -85,B 0,C 180,E1 -11378.274,E2 -11378.274} C_VEL
LIN {X 0,Y 397.144,Z 254.012,A -85,B 0,C 180,E1 -11381.993,E2 -11381.993} C_VEL
LIN {X 0,Y 397.101,Z 254.021,A -85,B 0,C 180,E1 -11385.064,E2 -11385.064} C_VEL
LIN {X 0,Y 397.055,Z 254.023,A -85,B 0,C 180,E1 -11388.02,E2 -11388.02} C_VEL
LIN {X 0,Y 397.12,Z 254.017,A -85,B 0,C 180,E1 -11391.138,E2 -11391.138} C_VEL
LIN {X 0,Y 397.108,Z 254.022,A -85,B 0,C 180,E1 -11394.496,E2 -11394.496} C_VEL
LIN {X 0,Y 397.066,Z 254.023,A -85,B 0,C 180,E1 -11397.928,E2 -11397.928} C_VEL
LIN {X 0,Y 397.109,Z 254.017,A -85,B 0,C 180,E1 -11401.456,E2 -11401.456} C_VEL
LIN {X 0,Y 397.112,Z 254.017,A -85,B 0,C 180,E1 -11403.741,E2 -11403.741} C_VEL
LIN {X 0,Y 396.993,Z 254.032,A -85,B 0,C 180,E1 -11407.079,E2 -11407.079} C_VEL
LIN {X 0,Y 396.87,Z 254.052,A -85,B 0,C 180,E1 -11408.169,E2 -11408.169} C_VEL
LIN {X 0,Y 396.881,Z 256.615,A -85,B 0,C 180,E1 -11410.34,E2 -11410.34} C_VEL
LIN {X 0,Y 396.742,Z 260.717,A -85,B 0,C 180,E1 -11413.535,E2 -11413.535} C_VEL
LIN {X 0,Y 396.612,Z 265.321,A -85,B 0,C 180,E1 -11417.052,E2 -11417.052} C_VEL
LIN {X 0,Y 396.411,Z 270.377,A -85,B 0,C 180,E1 -11420.819,E2 -11420.819} C_VEL
LIN {X 0,Y 396.377,Z 274.563,A -85,B 0,C 180,E1 -11423.893,E2 -11423.893} C_VEL
LIN {X 0,Y 396.337,Z 276.543,A -85,B 0,C 180,E1 -11425.328,E2 -11425.328} C_VEL
LIN {X 0,Y 398.867,Z 289.892,A -85,B 0,C 180,E1 -11425.879,E2 -11425.879} C_VEL
LIN {X 0,Y 400.958,Z 301.653,A -85,B 0,C 180,E1 -11426.546,E2 -11426.546} C_VEL
LIN {X 0,Y 400.267,Z 314.081,A -85,B 0,C 180,E1 -11427.358,E2 -11427.358} C_VEL
LIN {X 0,Y 399.486,Z 325.717,A -85,B 0,C 180,E1 -11428.362,E2 -11428.362} C_VEL
LIN {X 0,Y 398.739,Z 336.166,A -85,B 0,C 180,E1 -11429.495,E2 -11429.495} C_VEL
LIN {X 0,Y 397.979,Z 345.611,A -85,B 0,C 180,E1 -11430.759,E2 -11430.759} C_VEL
LIN {X 0,Y 397.198,Z 354.711,A -85,B 0,C 180,E1 -11432.282,E2 -11432.282} C_VEL
LIN {X 0,Y 396.71,Z 362.033,A -85,B 0,C 180,E1 -11433.809,E2 -11433.809} C_VEL
LIN {X 0,Y 396.331,Z 367.016,A -85,B 0,C 180,E1 -11435.087,E2 -11435.087} C_VEL
LIN {X 0,Y 396.16,Z 371.708,A -85,B 0,C 180,E1 -11436.574,E2 -11436.574} C_VEL
LIN {X 0,Y 395.903,Z 375.571,A -85,B 0,C 180,E1 -11438.164,E2 -11438.164} C_VEL
LIN {X 0,Y 395.763,Z 377.501,A -85,B 0,C 180,E1 -11439.196,E2 -11439.196} C_VEL
LIN {X 0,Y 395.69,Z 378.978,A -85,B 0,C 180,E1 -11440.231,E2 -11440.231} C_VEL
LIN {X 0,Y 395.684,Z 380.015,A -85,B 0,C 180,E1 -11441.266,E2 -11441.266} C_VEL
LIN {X 0,Y 395.697,Z 380.684,A -85,B 0,C 180,E1 -11442.358,E2 -11442.358} C_VEL
LIN {X 0,Y 395.612,Z 380.912,A -85,B 0,C 180,E1 -11443.352,E2 -11443.352} C_VEL
LIN {X 0,Y 395.609,Z 380.601,A -85,B 0,C 180,E1 -11444.593,E2 -11444.593} C_VEL
LIN {X 0,Y 395.772,Z 379.078,A -85,B 0,C 180,E1 -11446.506,E2 -11446.506} C_VEL
LIN {X 0,Y 395.863,Z 377.614,A -85,B 0,C 180,E1 -11447.566,E2 -11447.566} C_VEL
LIN {X 0,Y 396.109,Z 375.007,A -85,B 0,C 180,E1 -11448.937,E2 -11448.937} C_VEL
LIN {X 0,Y 395.611,Z 373.219,A -85,B 0,C 180,E1 -11449.75,E2 -11449.75} C_VEL
LIN {X 0,Y 393.083,Z 369.943,A -85,B 0,C 180,E1 -11451.062,E2 -11451.062} C_VEL
LIN {X 0,Y 390.634,Z 365.95,A -85,B 0,C 180,E1 -11452.343,E2 -11452.343} C_VEL
LIN {X 0,Y 390.261,Z 363.039,A -85,B 0,C 180,E1 -11453.098,E2 -11453.098} C_VEL
LIN {X 0,Y 391.033,Z 355.707,A -85,B 0,C 180,E1 -11454.7,E2 -11454.7} C_VEL
LIN {X 0,Y 391.966,Z 347.223,A -85,B 0,C 180,E1 -11456.189,E2 -11456.189} C_VEL
LIN {X 0,Y 392.959,Z 337.526,A -85,B 0,C 180,E1 -11457.565,E2 -11457.565} C_VEL
LIN {X 0,Y 393.995,Z 326.649,A -85,B 0,C 180,E1 -11458.79,E2 -11458.79} C_VEL
LIN {X 0,Y 394.909,Z 315.756,A -85,B 0,C 180,E1 -11459.77,E2 -11459.77} C_VEL
LIN {X 0,Y 395.762,Z 305.507,A -85,B 0,C 180,E1 -11460.493,E2 -11460.493} C_VEL
LIN {X 0,Y 394.603,Z 297.694,A -85,B 0,C 180,E1 -11461.034,E2 -11461.034} C_VEL
LIN {X 0,Y 391.609,Z 285.365,A -85,B 0,C 180,E1 -11461.781,E2 -11461.781} C_VEL
LIN {X 0,Y 389.192,Z 277.012,A -85,B 0,C 180,E1 -11462.226,E2 -11462.226} C_VEL
LIN {X 0,Y 389.385,Z 272.571,A -85,B 0,C 180,E1 -11465.691,E2 -11465.691} C_VEL
LIN {X 0,Y 389.628,Z 268.283,A -85,B 0,C 180,E1 -11469.146,E2 -11469.146} C_VEL
LIN {X 0,Y 389.897,Z 263.388,A -85,B 0,C 180,E1 -11473.231,E2 -11473.231} C_VEL
LIN {X 0,Y 390.123,Z 260.057,A -85,B 0,C 180,E1 -11476.102,E2 -11476.102} C_VEL
LIN {X 0,Y 390.202,Z 256.673,A -85,B 0,C 180,E1 -11479.152,E2 -11479.152} C_VEL
LIN {X 0,Y 390.056,Z 254.905,A -85,B 0,C 180,E1 -11480.906,E2 -11480.906} C_VEL
LIN {X 0,Y 390.073,Z 254.899,A -85,B 0,C 180,E1 -11484.794,E2 -11484.794} C_VEL
LIN {X 0,Y 390.015,Z 254.907,A -85,B 0,C 180,E1 -11488.497,E2 -11488.497} C_VEL
LIN {X 0,Y 390.106,Z 254.893,A -85,B 0,C 180,E1 -11492.071,E2 -11492.071} C_VEL
LIN {X 0,Y 390.07,Z 254.897,A -85,B 0,C 180,E1 -11495.52,E2 -11495.52} C_VEL
LIN {X 0,Y 390.092,Z 254.894,A -85,B 0,C 180,E1 -11498.881,E2 -11498.881} C_VEL
LIN {X 0,Y 390.12,Z 254.889,A -85,B 0,C 180,E1 -11502.168,E2 -11502.168} C_VEL
LIN {X 0,Y 390.135,Z 254.886,A -85,B 0,C 180,E1 -11505.394,E2 -11505.394} C_VEL
LIN {X 0,Y 390.138,Z 254.89,A -85,B 0,C 180,E1 -11508.572,E2 -11508.572} C_VEL
LIN {X 0,Y 390.298,Z 254.868,A -85,B 0,C 180,E1 -11512.032,E2 -11512.032} C_VEL
LIN {X 0,Y 390.216,Z 254.879,A -85,B 0,C 180,E1 -11514.835,E2 -11514.835} C_VEL
LIN {X 0,Y 390.412,Z 254.854,A -85,B 0,C 180,E1 -11517.938,E2 -11517.938} C_VEL
LIN {X 0,Y 390.537,Z 254.837,A -85,B 0,C 180,E1 -11520.001,E2 -11520.001} C_VEL
LIN {X 0,Y 390.307,Z 254.868,A -85,B 0,C 180,E1 -11523.098,E2 -11523.098} C_VEL
LIN {X 0,Y 390.319,Z 254.865,A -85,B 0,C 180,E1 -11526.203,E2 -11526.203} C_VEL
LIN {X 0,Y 390.307,Z 254.869,A -85,B 0,C 180,E1 -11528.283,E2 -11528.283} C_VEL
LIN {X 0,Y 390.164,Z 254.887,A -85,B 0,C 180,E1 -11532.484,E2 -11532.484} C_VEL
LIN {X 0,Y 390.132,Z 254.892,A -85,B 0,C 180,E1 -11535.678,E2 -11535.678} C_VEL
LIN {X 0,Y 390.099,Z 254.896,A -85,B 0,C 180,E1 -11538.923,E2 -11538.923} C_VEL
LIN {X 0,Y 390.034,Z 254.904,A -85,B 0,C 180,E1 -11542.236,E2 -11542.236} C_VEL
LIN {X 0,Y 390.106,Z 254.897,A -85,B 0,C 180,E1 -11545.742,E2 -11545.742} C_VEL
LIN {X 0,Y 390.04,Z 254.905,A -85,B 0,C 180,E1 -11549.112,E2 -11549.112} C_VEL
LIN {X 0,Y 390.039,Z 254.902,A -85,B 0,C 180,E1 -11552.723,E2 -11552.723} C_VEL
LIN {X 0,Y 390.053,Z 254.899,A -85,B 0,C 180,E1 -11555.827,E2 -11555.827} C_VEL
LIN {X 0,Y 390.067,Z 254.896,A -85,B 0,C 180,E1 -11559.22,E2 -11559.22} C_VEL
LIN {X 0,Y 390.04,Z 254.898,A -85,B 0,C 180,E1 -11562.375,E2 -11562.375} C_VEL
LIN {X 0,Y 390.041,Z 254.894,A -85,B 0,C 180,E1 -11565.355,E2 -11565.355} C_VEL
LIN {X 0,Y 390.06,Z 254.937,A -85,B 0,C 180,E1 -11566.455,E2 -11566.455} C_VEL
LIN {X 0,Y 390.795,Z 259.32,A -85,B 0,C 180,E1 -11569.654,E2 -11569.654} C_VEL
LIN {X 0,Y 391.52,Z 264.323,A -85,B 0,C 180,E1 -11573.035,E2 -11573.035} C_VEL
LIN {X 0,Y 391.541,Z 268.505,A -85,B 0,C 180,E1 -11575.659,E2 -11575.659} C_VEL
LIN {X 0,Y 391.061,Z 273.491,A -85,B 0,C 180,E1 -11578.59,E2 -11578.59} C_VEL
LIN {X 0,Y 390.455,Z 279.319,A -85,B 0,C 180,E1 -11581.883,E2 -11581.883} C_VEL
LIN {X 0,Y 389.985,Z 285.965,A -85,B 0,C 180,E1 -11585.514,E2 -11585.514} C_VEL
LIN {X 0,Y 389.614,Z 292.272,A -85,B 0,C 180,E1 -11588.853,E2 -11588.853} C_VEL
LIN {X 0,Y 389.37,Z 296.084,A -85,B 0,C 180,E1 -11590.836,E2 -11590.836} C_VEL
LIN {X 0,Y 392.387,Z 309.188,A -85,B 0,C 180,E1 -11591.449,E2 -11591.449} C_VEL
LIN {X 0,Y 394.276,Z 320.834,A -85,B 0,C 180,E1 -11592.136,E2 -11592.136} C_VEL
LIN {X 0,Y 395.004,Z 328.485,A -85,B 0,C 180,E1 -11592.662,E2 -11592.662} C_VEL
LIN {X 0,Y 394.047,Z 340.382,A -85,B 0,C 180,E1 -11593.553,E2 -11593.553} C_VEL
LIN {X 0,Y 393.012,Z 351.033,A -85,B 0,C 180,E1 -11594.574,E2 -11594.574} C_VEL
LIN {X 0,Y 392.097,Z 360.808,A -85,B 0,C 180,E1 -11595.74,E2 -11595.74} C_VEL
LIN {X 0,Y 391.291,Z 369.623,A -85,B 0,C 180,E1 -11597.026,E2 -11597.026} C_VEL
LIN {X 0,Y 390.252,Z 378.313,A -85,B 0,C 180,E1 -11598.575,E2 -11598.575} C_VEL
LIN {X 0,Y 389.657,Z 385.265,A -85,B 0,C 180,E1 -11600.134,E2 -11600.134} C_VEL
LIN {X 0,Y 389.203,Z 390.852,A -85,B 0,C 180,E1 -11601.694,E2 -11601.694} C_VEL
LIN {X 0,Y 388.878,Z 395.259,A -85,B 0,C 180,E1 -11603.254,E2 -11603.254} C_VEL
LIN {X 0,Y 388.743,Z 398.606,A -85,B 0,C 180,E1 -11604.814,E2 -11604.814} C_VEL
LIN {X 0,Y 388.701,Z 400.277,A -85,B 0,C 180,E1 -11605.853,E2 -11605.853} C_VEL
LIN {X 0,Y 388.661,Z 402.427,A -85,B 0,C 180,E1 -11607.928,E2 -11607.928} C_VEL
LIN {X 0,Y 388.704,Z 402.871,A -85,B 0,C 180,E1 -11608.964,E2 -11608.964} C_VEL
LIN {X 0,Y 388.709,Z 402.922,A -85,B 0,C 180,E1 -11610,E2 -11610} C_VEL
LIN {X 0,Y 388.705,Z 402.587,A -85,B 0,C 180,E1 -11611.036,E2 -11611.036} C_VEL
LIN {X 0,Y 388.678,Z 401.863,A -85,B 0,C 180,E1 -11612.072,E2 -11612.072} C_VEL
LIN {X 0,Y 388.639,Z 400.697,A -85,B 0,C 180,E1 -11613.11,E2 -11613.11} C_VEL
LIN {X 0,Y 388.714,Z 398.183,A -85,B 0,C 180,E1 -11614.667,E2 -11614.667} C_VEL
LIN {X 0,Y 388.798,Z 394.646,A -85,B 0,C 180,E1 -11616.226,E2 -11616.226} C_VEL
LIN {X 0,Y 389.002,Z 389.994,A -85,B 0,C 180,E1 -11617.787,E2 -11617.787} C_VEL
LIN {X 0,Y 389.45,Z 382.958,A -85,B 0,C 180,E1 -11619.609,E2 -11619.609} C_VEL
LIN {X 0,Y 389.936,Z 375.324,A -85,B 0,C 180,E1 -11621.172,E2 -11621.172} C_VEL
LIN {X 0,Y 390.647,Z 367.522,A -85,B 0,C 180,E1 -11622.467,E2 -11622.467} C_VEL
LIN {X 0,Y 391.402,Z 357.269,A -85,B 0,C 180,E1 -11623.849,E2 -11623.849} C_VEL
LIN {X 0,Y 392.203,Z 346.053,A -85,B 0,C 180,E1 -11625.06,E2 -11625.06} C_VEL
LIN {X 0,Y 392.97,Z 335.52,A -85,B 0,C 180,E1 -11625.96,E2 -11625.96} C_VEL
LIN {X 0,Y 393.426,Z 326.112,A -85,B 0,C 180,E1 -11626.607,E2 -11626.607} C_VEL
LIN {X 0,Y 391.83,Z 313.42,A -85,B 0,C 180,E1 -11627.35,E2 -11627.35} C_VEL
LIN {X 0,Y 389.586,Z 299.369,A -85,B 0,C 180,E1 -11627.947,E2 -11627.947} C_VEL
LIN {X 0,Y 389.129,Z 296.384,A -85,B 0,C 180,E1 -11628.05,E2 -11628.05} C_VEL
LIN {X 0,Y 389.437,Z 290.18,A -85,B 0,C 180,E1 -11631.157,E2 -11631.157} C_VEL
LIN {X 0,Y 389.723,Z 283.591,A -85,B 0,C 180,E1 -11634.504,E2 -11634.504} C_VEL
LIN {X 0,Y 390.146,Z 277.006,A -85,B 0,C 180,E1 -11637.927,E2 -11637.927} C_VEL
LIN {X 0,Y 390.543,Z 271.494,A -85,B 0,C 180,E1 -11640.854,E2 -11640.854} C_VEL
LIN {X 0,Y 391.029,Z 265.314,A -85,B 0,C 180,E1 -11644.231,E2 -11644.231} C_VEL
LIN {X 0,Y 391.076,Z 261.537,A -85,B 0,C 180,E1 -11646.372,E2 -11646.372} C_VEL
LIN {X 0,Y 390.414,Z 256.694,A -85,B 0,C 180,E1 -11649.279,E2 -11649.279} C_VEL
LIN {X 0,Y 390.087,Z 254.896,A -85,B 0,C 180,E1 -11650.435,E2 -11650.435} C_VEL
LIN {X 0,Y 390.022,Z 254.899,A -85,B 0,C 180,E1 -11653.88,E2 -11653.88} C_VEL
LIN {X 0,Y 390.004,Z 254.902,A -85,B 0,C 180,E1 -11657.631,E2 -11657.631} C_VEL
LIN {X 0,Y 390.054,Z 254.9,A -85,B 0,C 180,E1 -11660.902,E2 -11660.902} C_VEL
LIN {X 0,Y 390.065,Z 254.898,A -85,B 0,C 180,E1 -11664.79,E2 -11664.79} C_VEL
LIN {X 0,Y 390.019,Z 254.905,A -85,B 0,C 180,E1 -11668.494,E2 -11668.494} C_VEL
LIN {X 0,Y 390.024,Z 254.902,A -85,B 0,C 180,E1 -11672.062,E2 -11672.062} C_VEL
LIN {X 0,Y 390.047,Z 254.897,A -85,B 0,C 180,E1 -11675.516,E2 -11675.516} C_VEL
LIN {X 0,Y 390.05,Z 254.899,A -85,B 0,C 180,E1 -11678.876,E2 -11678.876} C_VEL
LIN {X 0,Y 390.122,Z 254.892,A -85,B 0,C 180,E1 -11682.165,E2 -11682.165} C_VEL
LIN {X 0,Y 390.137,Z 254.886,A -85,B 0,C 180,E1 -11685.391,E2 -11685.391} C_VEL
LIN {X 0,Y 390.141,Z 254.888,A -85,B 0,C 180,E1 -11688.57,E2 -11688.57} C_VEL
LIN {X 0,Y 390.301,Z 254.869,A -85,B 0,C 180,E1 -11692.03,E2 -11692.03} C_VEL
LIN {X 0,Y 390.218,Z 254.876,A -85,B 0,C 180,E1 -11694.832,E2 -11694.832} C_VEL
LIN {X 0,Y 390.412,Z 254.855,A -85,B 0,C 180,E1 -11697.936,E2 -11697.936} C_VEL
LIN {X 0,Y 390.543,Z 254.839,A -85,B 0,C 180,E1 -11699.999,E2 -11699.999} C_VEL
LIN {X 0,Y 390.308,Z 254.865,A -85,B 0,C 180,E1 -11703.095,E2 -11703.095} C_VEL
LIN {X 0,Y 390.301,Z 254.866,A -85,B 0,C 180,E1 -11706.658,E2 -11706.658} C_VEL
LIN {X 0,Y 390.196,Z 254.881,A -85,B 0,C 180,E1 -11709.328,E2 -11709.328} C_VEL
LIN {X 0,Y 390.161,Z 254.883,A -85,B 0,C 180,E1 -11712.482,E2 -11712.482} C_VEL
LIN {X 0,Y 390.129,Z 254.891,A -85,B 0,C 180,E1 -11715.676,E2 -11715.676} C_VEL
LIN {X 0,Y 390.095,Z 254.893,A -85,B 0,C 180,E1 -11718.921,E2 -11718.921} C_VEL
LIN {X 0,Y 390.029,Z 254.899,A -85,B 0,C 180,E1 -11722.233,E2 -11722.233} C_VEL
LIN {X 0,Y 390.108,Z 254.891,A -85,B 0,C 180,E1 -11725.743,E2 -11725.743} C_VEL
LIN {X 0,Y 390.054,Z 254.9,A -85,B 0,C 180,E1 -11729.108,E2 -11729.108} C_VEL
LIN {X 0,Y 390.032,Z 254.9,A -85,B 0,C 180,E1 -11732.721,E2 -11732.721} C_VEL
LIN {X 0,Y 390.046,Z 254.897,A -85,B 0,C 180,E1 -11735.825,E2 -11735.825} C_VEL
LIN {X 0,Y 390.063,Z 254.898,A -85,B 0,C 180,E1 -11739.219,E2 -11739.219} C_VEL
LIN {X 0,Y 390.108,Z 254.89,A -85,B 0,C 180,E1 -11742.386,E2 -11742.386} C_VEL
LIN {X 0,Y 390.051,Z 254.896,A -85,B 0,C 180,E1 -11745.357,E2 -11745.357} C_VEL
LIN {X 0,Y 390.02,Z 254.9,A -85,B 0,C 180,E1 -11748.186,E2 -11748.186} C_VEL
LIN {X 0,Y 390.079,Z 254.896,A -85,B 0,C 180,E1 -11750.907,E2 -11750.907} C_VEL
LIN {X 0,Y 390.073,Z 254.896,A -85,B 0,C 180,E1 -11754.793,E2 -11754.793} C_VEL
LIN {X 0,Y 390.012,Z 254.906,A -85,B 0,C 180,E1 -11758.495,E2 -11758.495} C_VEL
LIN {X 0,Y 390.106,Z 254.892,A -85,B 0,C 180,E1 -11762.07,E2 -11762.07} C_VEL
LIN {X 0,Y 390.069,Z 254.898,A -85,B 0,C 180,E1 -11764.38,E2 -11764.38} C_VEL
LIN {X 0,Y 389.855,Z 254.922,A -85,B 0,C 180,E1 -11767.755,E2 -11767.755} C_VEL
LIN {X 0,Y 389.801,Z 255.645,A -85,B 0,C 180,E1 -11768.864,E2 -11768.864} C_VEL
LIN {X 0,Y 389.78,Z 258.373,A -85,B 0,C 180,E1 -11771.062,E2 -11771.062} C_VEL
LIN {X 0,Y 389.59,Z 262.48,A -85,B 0,C 180,E1 -11774.301,E2 -11774.301} C_VEL
LIN {X 0,Y 389.511,Z 266.618,A -85,B 0,C 180,E1 -11777.496,E2 -11777.496} C_VEL
LIN {X 0,Y 389.349,Z 270.789,A -85,B 0,C 180,E1 -11780.651,E2 -11780.651} C_VEL
LIN {X 0,Y 389.331,Z 275.003,A -85,B 0,C 180,E1 -11783.782,E2 -11783.782} C_VEL
LIN {X 0,Y 389.247,Z 276.74,A -85,B 0,C 180,E1 -11785.048,E2 -11785.048} C_VEL
LIN {X 0,Y 391.891,Z 290.27,A -85,B 0,C 180,E1 -11785.629,E2 -11785.629} C_VEL
LIN {X 0,Y 394.007,Z 302.783,A -85,B 0,C 180,E1 -11786.357,E2 -11786.357} C_VEL
LIN {X 0,Y 393.306,Z 314.939,A -85,B 0,C 180,E1 -11787.183,E2 -11787.183} C_VEL
LIN {X 0,Y 392.513,Z 326.445,A -85,B 0,C 180,E1 -11788.204,E2 -11788.204} C_VEL
LIN {X 0,Y 391.738,Z 336.811,A -85,B 0,C 180,E1 -11789.358,E2 -11789.358} C_VEL
LIN {X 0,Y 390.996,Z 345.312,A -85,B 0,C 180,E1 -11790.515,E2 -11790.515} C_VEL
LIN {X 0,Y 390.332,Z 353.151,A -85,B 0,C 180,E1 -11791.806,E2 -11791.806} C_VEL
LIN {X 0,Y 389.761,Z 360.803,A -85,B 0,C 180,E1 -11793.359,E2 -11793.359} C_VEL
LIN {X 0,Y 389.248,Z 367.867,A -85,B 0,C 180,E1 -11795.179,E2 -11795.179} C_VEL
LIN {X 0,Y 389.076,Z 372.061,A -85,B 0,C 180,E1 -11796.561,E2 -11796.561} C_VEL
LIN {X 0,Y 388.801,Z 376.161,A -85,B 0,C 180,E1 -11798.314,E2 -11798.314} C_VEL
LIN {X 0,Y 388.659,Z 378.007,A -85,B 0,C 180,E1 -11799.366,E2 -11799.366} C_VEL
LIN {X 0,Y 388.607,Z 379.385,A -85,B 0,C 180,E1 -11800.419,E2 -11800.419} C_VEL
LIN {X 0,Y 388.605,Z 380.9,A -85,B 0,C 180,E1 -11802.428,E2 -11802.428} C_VEL
LIN {X 0,Y 388.529,Z 381.099,A -85,B 0,C 180,E1 -11803.6,E2 -11803.6} C_VEL
LIN {X 0,Y 388.519,Z 380.826,A -85,B 0,C 180,E1 -11804.669,E2 -11804.669} C_VEL
LIN {X 0,Y 388.697,Z 379.287,A -85,B 0,C 180,E1 -11806.613,E2 -11806.613} C_VEL
LIN {X 0,Y 388.931,Z 376.561,A -85,B 0,C 180,E1 -11808.434,E2 -11808.434} C_VEL
LIN {X 0,Y 389.292,Z 372.72,A -85,B 0,C 180,E1 -11810.159,E2 -11810.159} C_VEL
LIN {X 0,Y 389.728,Z 368.196,A -85,B 0,C 180,E1 -11811.695,E2 -11811.695} C_VEL
LIN {X 0,Y 390.261,Z 363.039,A -85,B 0,C 180,E1 -11813.098,E2 -11813.098} C_VEL
LIN {X 0,Y 389.933,Z 359.999,A -85,B 0,C 180,E1 -11813.837,E2 -11813.837} C_VEL
LIN {X 0,Y 387.733,Z 354.76,A -85,B 0,C 180,E1 -11815.042,E2 -11815.042} C_VEL
LIN {X 0,Y 385.604,Z 349.034,A -85,B 0,C 180,E1 -11816.198,E2 -11816.198} C_VEL
LIN {X 0,Y 385.379,Z 345.089,A -85,B 0,C 180,E1 -11816.849,E2 -11816.849} C_VEL
LIN {X 0,Y 386.424,Z 335.03,A -85,B 0,C 180,E1 -11818.22,E2 -11818.22} C_VEL
LIN {X 0,Y 387.473,Z 324.966,A -85,B 0,C 180,E1 -11819.322,E2 -11819.322} C_VEL
LIN {X 0,Y 388.443,Z 314.045,A -85,B 0,C 180,E1 -11820.277,E2 -11820.277} C_VEL
LIN {X 0,Y 389,Z 305.159,A -85,B 0,C 180,E1 -11820.908,E2 -11820.908} C_VEL
LIN {X 0,Y 386.871,Z 294.1,A -85,B 0,C 180,E1 -11821.687,E2 -11821.687} C_VEL
LIN {X 0,Y 383.447,Z 281.909,A -85,B 0,C 180,E1 -11822.411,E2 -11822.411} C_VEL
LIN {X 0,Y 382.15,Z 277.202,A -85,B 0,C 180,E1 -11822.674,E2 -11822.674} C_VEL
LIN {X 0,Y 382.352,Z 272.992,A -85,B 0,C 180,E1 -11826.028,E2 -11826.028} C_VEL
LIN {X 0,Y 382.579,Z 268.744,A -85,B 0,C 180,E1 -11829.51,E2 -11829.51} C_VEL
LIN {X 0,Y 382.83,Z 264.888,A -85,B 0,C 180,E1 -11832.783,E2 -11832.783} C_VEL
LIN {X 0,Y 383.068,Z 261.435,A -85,B 0,C 180,E1 -11835.802,E2 -11835.802} C_VEL
LIN {X 0,Y 383.19,Z 258.188,A -85,B 0,C 180,E1 -11838.76,E2 -11838.76} C_VEL
LIN {X 0,Y 383.052,Z 256.475,A -85,B 0,C 180,E1 -11840.405,E2 -11840.405} C_VEL
LIN {X 0,Y 382.977,Z 255.785,A -85,B 0,C 180,E1 -11841.398,E2 -11841.398} C_VEL
LIN {X 0,Y 383.013,Z 255.778,A -85,B 0,C 180,E1 -11844.045,E2 -11844.045} C_VEL
LIN {X 0,Y 382.976,Z 255.785,A -85,B 0,C 180,E1 -11847.578,E2 -11847.578} C_VEL
LIN {X 0,Y 382.986,Z 255.783,A -85,B 0,C 180,E1 -11850.301,E2 -11850.301} C_VEL
LIN {X 0,Y 383.045,Z 255.771,A -85,B 0,C 180,E1 -11852.699,E2 -11852.699} C_VEL
LIN {X 0,Y 383.031,Z 255.776,A -85,B 0,C 180,E1 -11856.194,E2 -11856.194} C_VEL
LIN {X 0,Y 383.071,Z 255.767,A -85,B 0,C 180,E1 -11859.601,E2 -11859.601} C_VEL
LIN {X 0,Y 383.096,Z 255.764,A -85,B 0,C 180,E1 -11862.932,E2 -11862.932} C_VEL
LIN {X 0,Y 383.115,Z 255.761,A -85,B 0,C 180,E1 -11866.465,E2 -11866.465} C_VEL
LIN {X 0,Y 383.142,Z 255.76,A -85,B 0,C 180,E1 -11870.499,E2 -11870.499} C_VEL
LIN {X 0,Y 383.246,Z 255.747,A -85,B 0,C 180,E1 -11872.626,E2 -11872.626} C_VEL
LIN {X 0,Y 383.188,Z 255.755,A -85,B 0,C 180,E1 -11874.74,E2 -11874.74} C_VEL
LIN {X 0,Y 383.379,Z 255.73,A -85,B 0,C 180,E1 -11877.9,E2 -11877.9} C_VEL
LIN {X 0,Y 383.507,Z 255.713,A -85,B 0,C 180,E1 -11880.001,E2 -11880.001} C_VEL
LIN {X 0,Y 383.244,Z 255.748,A -85,B 0,C 180,E1 -11883.155,E2 -11883.155} C_VEL
LIN {X 0,Y 383.276,Z 255.743,A -85,B 0,C 180,E1 -11886.318,E2 -11886.318} C_VEL
LIN {X 0,Y 383.253,Z 255.746,A -85,B 0,C 180,E1 -11888.437,E2 -11888.437} C_VEL
LIN {X 0,Y 383.09,Z 255.765,A -85,B 0,C 180,E1 -11891.643,E2 -11891.643} C_VEL
LIN {X 0,Y 383.103,Z 255.765,A -85,B 0,C 180,E1 -11894.883,E2 -11894.883} C_VEL
LIN {X 0,Y 383.083,Z 255.77,A -85,B 0,C 180,E1 -11898.174,E2 -11898.174} C_VEL
LIN {X 0,Y 382.987,Z 255.784,A -85,B 0,C 180,E1 -11901.532,E2 -11901.532} C_VEL
LIN {X 0,Y 383.043,Z 255.777,A -85,B 0,C 180,E1 -11904.962,E2 -11904.962} C_VEL
LIN {X 0,Y 382.998,Z 255.781,A -85,B 0,C 180,E1 -11908.497,E2 -11908.497} C_VEL
LIN {X 0,Y 383.006,Z 255.78,A -85,B 0,C 180,E1 -11912.151,E2 -11912.151} C_VEL
LIN {X 0,Y 383.015,Z 255.777,A -85,B 0,C 180,E1 -11914.669,E2 -11914.669} C_VEL
LIN {X 0,Y 382.997,Z 255.778,A -85,B 0,C 180,E1 -11917.905,E2 -11917.905} C_VEL
LIN {X 0,Y 382.982,Z 255.78,A -85,B 0,C 180,E1 -11921.349,E2 -11921.349} C_VEL
LIN {X 0,Y 382.994,Z 255.77,A -85,B 0,C 180,E1 -11924.304,E2 -11924.304} C_VEL
LIN {X 0,Y 383.034,Z 255.872,A -85,B 0,C 180,E1 -11926.075,E2 -11926.075} C_VEL
LIN {X 0,Y 383.606,Z 259.396,A -85,B 0,C 180,E1 -11928.736,E2 -11928.736} C_VEL
LIN {X 0,Y 384.324,Z 263.788,A -85,B 0,C 180,E1 -11931.845,E2 -11931.845} C_VEL
LIN {X 0,Y 384.592,Z 267.387,A -85,B 0,C 180,E1 -11934.215,E2 -11934.215} C_VEL
LIN {X 0,Y 384.342,Z 271.442,A -85,B 0,C 180,E1 -11936.732,E2 -11936.732} C_VEL
LIN {X 0,Y 383.898,Z 275.903,A -85,B 0,C 180,E1 -11939.366,E2 -11939.366} C_VEL
LIN {X 0,Y 383.202,Z 282.806,A -85,B 0,C 180,E1 -11943.3,E2 -11943.3} C_VEL
LIN {X 0,Y 382.82,Z 288.838,A -85,B 0,C 180,E1 -11946.626,E2 -11946.626} C_VEL
LIN {X 0,Y 382.366,Z 295.366,A -85,B 0,C 180,E1 -11950.121,E2 -11950.121} C_VEL
LIN {X 0,Y 382.322,Z 295.891,A -85,B 0,C 180,E1 -11950.399,E2 -11950.399} C_VEL
LIN {X 0,Y 385.531,Z 309.48,A -85,B 0,C 180,E1 -11951.063,E2 -11951.063} C_VEL
LIN {X 0,Y 387.482,Z 321.431,A -85,B 0,C 180,E1 -11951.798,E2 -11951.798} C_VEL
LIN {X 0,Y 388.192,Z 331.003,A -85,B 0,C 180,E1 -11952.484,E2 -11952.484} C_VEL
LIN {X 0,Y 387.154,Z 342.219,A -85,B 0,C 180,E1 -11953.387,E2 -11953.387} C_VEL
LIN {X 0,Y 385.924,Z 353.661,A -85,B 0,C 180,E1 -11954.555,E2 -11954.555} C_VEL
LIN {X 0,Y 385.022,Z 363.327,A -85,B 0,C 180,E1 -11955.798,E2 -11955.798} C_VEL
LIN {X 0,Y 383.991,Z 372.829,A -85,B 0,C 180,E1 -11957.313,E2 -11957.313} C_VEL
LIN {X 0,Y 383.061,Z 380.836,A -85,B 0,C 180,E1 -11958.893,E2 -11958.893} C_VEL
LIN {X 0,Y 382.449,Z 387.284,A -85,B 0,C 180,E1 -11960.481,E2 -11960.481} C_VEL
LIN {X 0,Y 382.045,Z 392.423,A -85,B 0,C 180,E1 -11962.07,E2 -11962.07} C_VEL
LIN {X 0,Y 381.698,Z 396.864,A -85,B 0,C 180,E1 -11963.872,E2 -11963.872} C_VEL
LIN {X 0,Y 381.626,Z 400.151,A -85,B 0,C 180,E1 -11965.776,E2 -11965.776} C_VEL
LIN {X 0,Y 381.546,Z 401.406,A -85,B 0,C 180,E1 -11966.832,E2 -11966.832} C_VEL
LIN {X 0,Y 381.559,Z 402.258,A -85,B 0,C 180,E1 -11967.889,E2 -11967.889} C_VEL
LIN {X 0,Y 381.604,Z 402.679,A -85,B 0,C 180,E1 -11968.945,E2 -11968.945} C_VEL
LIN {X 0,Y 381.64,Z 402.714,A -85,B 0,C 180,E1 -11970,E2 -11970} C_VEL
LIN {X 0,Y 381.62,Z 402.363,A -85,B 0,C 180,E1 -11971.055,E2 -11971.055} C_VEL
LIN {X 0,Y 381.577,Z 401.616,A -85,B 0,C 180,E1 -11972.111,E2 -11972.111} C_VEL
LIN {X 0,Y 381.55,Z 400.424,A -85,B 0,C 180,E1 -11973.168,E2 -11973.168} C_VEL
LIN {X 0,Y 381.632,Z 397.875,A -85,B 0,C 180,E1 -11974.754,E2 -11974.754} C_VEL
LIN {X 0,Y 381.713,Z 394.3,A -85,B 0,C 180,E1 -11976.342,E2 -11976.342} C_VEL
LIN {X 0,Y 381.929,Z 389.605,A -85,B 0,C 180,E1 -11977.933,E2 -11977.933} C_VEL
LIN {X 0,Y 382.4,Z 382.521,A -85,B 0,C 180,E1 -11979.788,E2 -11979.788} C_VEL
LIN {X 0,Y 382.935,Z 374.831,A -85,B 0,C 180,E1 -11981.379,E2 -11981.379} C_VEL
LIN {X 0,Y 383.654,Z 366.954,A -85,B 0,C 180,E1 -11982.698,E2 -11982.698} C_VEL
LIN {X 0,Y 384.376,Z 357.631,A -85,B 0,C 180,E1 -11983.98,E2 -11983.98} C_VEL
LIN {X 0,Y 385.193,Z 346.608,A -85,B 0,C 180,E1 -11985.205,E2 -11985.205} C_VEL
LIN {X 0,Y 385.997,Z 336.273,A -85,B 0,C 180,E1 -11986.12,E2 -11986.12} C_VEL
LIN {X 0,Y 386.511,Z 327.082,A -85,B 0,C 180,E1 -11986.777,E2 -11986.777} C_VEL
LIN {X 0,Y 385.026,Z 315.085,A -85,B 0,C 180,E1 -11987.523,E2 -11987.523} C_VEL
LIN {X 0,Y 383.052,Z 302.228,A -85,B 0,C 180,E1 -11988.117,E2 -11988.117} C_VEL
LIN {X 0,Y 382.093,Z 296.198,A -85,B 0,C 180,E1 -11988.325,E2 -11988.325} C_VEL
LIN {X 0,Y 382.445,Z 288.776,A -85,B 0,C 180,E1 -11992.13,E2 -11992.13} C_VEL
LIN {X 0,Y 382.87,Z 281.545,A -85,B 0,C 180,E1 -11995.913,E2 -11995.913} C_VEL
LIN {X 0,Y 383.341,Z 274.505,A -85,B 0,C 180,E1 -11999.669,E2 -11999.669} C_VEL
LIN {X 0,Y 383.863,Z 267.91,A -85,B 0,C 180,E1 -12003.315,E2 -12003.315} C_VEL
LIN {X 0,Y 384.113,Z 263.47,A -85,B 0,C 180,E1 -12005.837,E2 -12005.837} C_VEL
LIN {X 0,Y 383.57,Z 259.023,A -85,B 0,C 180,E1 -12008.532,E2 -12008.532} C_VEL
LIN {X 0,Y 383.033,Z 255.775,A -85,B 0,C 180,E1 -12010.643,E2 -12010.643} C_VEL
LIN {X 0,Y 382.991,Z 255.776,A -85,B 0,C 180,E1 -12014.301,E2 -12014.301} C_VEL
LIN {X 0,Y 382.974,Z 255.78,A -85,B 0,C 180,E1 -12017.234,E2 -12017.234} C_VEL
LIN {X 0,Y 382.982,Z 255.779,A -85,B 0,C 180,E1 -12020.418,E2 -12020.418} C_VEL
LIN {X 0,Y 383.009,Z 255.774,A -85,B 0,C 180,E1 -12024.042,E2 -12024.042} C_VEL
LIN {X 0,Y 382.982,Z 255.777,A -85,B 0,C 180,E1 -12027.577,E2 -12027.577} C_VEL
LIN {X 0,Y 382.974,Z 255.781,A -85,B 0,C 180,E1 -12030.297,E2 -12030.297} C_VEL
LIN {X 0,Y 382.999,Z 255.777,A -85,B 0,C 180,E1 -12034.043,E2 -12034.043} C_VEL
LIN {X 0,Y 382.985,Z 255.777,A -85,B 0,C 180,E1 -12037.333,E2 -12037.333} C_VEL
LIN {X 0,Y 383.054,Z 255.771,A -85,B 0,C 180,E1 -12040.715,E2 -12040.715} C_VEL
LIN {X 0,Y 383.074,Z 255.77,A -85,B 0,C 180,E1 -12044.025,E2 -12044.025} C_VEL
LIN {X 0,Y 383.13,Z 255.759,A -85,B 0,C 180,E1 -12047.283,E2 -12047.283} C_VEL
LIN {X 0,Y 383.144,Z 255.76,A -85,B 0,C 180,E1 -12050.497,E2 -12050.497} C_VEL
LIN {X 0,Y 383.275,Z 255.743,A -85,B 0,C 180,E1 -12053.682,E2 -12053.682} C_VEL
LIN {X 0,Y 383.379,Z 255.731,A -85,B 0,C 180,E1 -12057.898,E2 -12057.898} C_VEL
LIN {X 0,Y 383.513,Z 255.715,A -85,B 0,C 180,E1 -12059.999,E2 -12059.999} C_VEL
LIN {X 0,Y 383.244,Z 255.745,A -85,B 0,C 180,E1 -12063.152,E2 -12063.152} C_VEL
LIN {X 0,Y 383.26,Z 255.742,A -85,B 0,C 180,E1 -12066.653,E2 -12066.653} C_VEL
LIN {X 0,Y 383.251,Z 255.744,A -85,B 0,C 180,E1 -12068.435,E2 -12068.435} C_VEL
LIN {X 0,Y 383.089,Z 255.768,A -85,B 0,C 180,E1 -12071.641,E2 -12071.641} C_VEL
LIN {X 0,Y 383.1,Z 255.763,A -85,B 0,C 180,E1 -12074.881,E2 -12074.881} C_VEL
LIN {X 0,Y 383.052,Z 255.769,A -85,B 0,C 180,E1 -12078.173,E2 -12078.173} C_VEL
LIN {X 0,Y 382.982,Z 255.782,A -85,B 0,C 180,E1 -12081.53,E2 -12081.53} C_VEL
LIN {X 0,Y 383.041,Z 255.772,A -85,B 0,C 180,E1 -12084.959,E2 -12084.959} C_VEL
LIN {X 0,Y 383.038,Z 255.77,A -85,B 0,C 180,E1 -12088.491,E2 -12088.491} C_VEL
LIN {X 0,Y 382.999,Z 255.774,A -85,B 0,C 180,E1 -12092.149,E2 -12092.149} C_VEL
LIN {X 0,Y 383.007,Z 255.775,A -85,B 0,C 180,E1 -12094.667,E2 -12094.667} C_VEL
LIN {X 0,Y 382.992,Z 255.775,A -85,B 0,C 180,E1 -12097.904,E2 -12097.904} C_VEL
LIN {X 0,Y 383.035,Z 255.772,A -85,B 0,C 180,E1 -12101.339,E2 -12101.339} C_VEL
LIN {X 0,Y 383.023,Z 255.772,A -85,B 0,C 180,E1 -12104.309,E2 -12104.309} C_VEL
LIN {X 0,Y 382.998,Z 255.776,A -85,B 0,C 180,E1 -12107.24,E2 -12107.24} C_VEL
LIN {X 0,Y 383.004,Z 255.776,A -85,B 0,C 180,E1 -12110.413,E2 -12110.413} C_VEL
LIN {X 0,Y 383.014,Z 255.773,A -85,B 0,C 180,E1 -12114.044,E2 -12114.044} C_VEL
LIN {X 0,Y 382.974,Z 255.777,A -85,B 0,C 180,E1 -12117.578,E2 -12117.578} C_VEL
LIN {X 0,Y 382.98,Z 255.781,A -85,B 0,C 180,E1 -12120.3,E2 -12120.3} C_VEL
LIN {X 0,Y 383.035,Z 255.771,A -85,B 0,C 180,E1 -12123.874,E2 -12123.874} C_VEL
LIN {X 0,Y 382.85,Z 255.793,A -85,B 0,C 180,E1 -12127.326,E2 -12127.326} C_VEL
LIN {X 0,Y 382.753,Z 256.029,A -85,B 0,C 180,E1 -12128.455,E2 -12128.455} C_VEL
LIN {X 0,Y 382.735,Z 258.744,A -85,B 0,C 180,E1 -12130.7,E2 -12130.7} C_VEL
LIN {X 0,Y 382.548,Z 262.875,A -85,B 0,C 180,E1 -12134.004,E2 -12134.004} C_VEL
LIN {X 0,Y 382.472,Z 267.027,A -85,B 0,C 180,E1 -12137.262,E2 -12137.262} C_VEL
LIN {X 0,Y 382.284,Z 272.623,A -85,B 0,C 180,E1 -12141.543,E2 -12141.543} C_VEL
LIN {X 0,Y 382.285,Z 275.441,A -85,B 0,C 180,E1 -12143.667,E2 -12143.667} C_VEL
LIN {X 0,Y 382.161,Z 276.908,A -85,B 0,C 180,E1 -12144.757,E2 -12144.757} C_VEL
LIN {X 0,Y 385.004,Z 290.962,A -85,B 0,C 180,E1 -12145.387,E2 -12145.387} C_VEL
LIN {X 0,Y 386.799,Z 301.852,A -85,B 0,C 180,E1 -12146.028,E2 -12146.028} C_VEL
LIN {X 0,Y 387.02,Z 304.922,A -85,B 0,C 180,E1 -12146.226,E2 -12146.226} C_VEL
LIN {X 0,Y 386.255,Z 317.354,A -85,B 0,C 180,E1 -12147.132,E2 -12147.132} C_VEL
LIN {X 0,Y 385.38,Z 328.475,A -85,B 0,C 180,E1 -12148.171,E2 -12148.171} C_VEL
LIN {X 0,Y 384.737,Z 337.448,A -85,B 0,C 180,E1 -12149.215,E2 -12149.215} C_VEL
LIN {X 0,Y 383.916,Z 346.701,A -85,B 0,C 180,E1 -12150.524,E2 -12150.524} C_VEL
LIN {X 0,Y 383.087,Z 355.682,A -85,B 0,C 180,E1 -12152.103,E2 -12152.103} C_VEL
LIN {X 0,Y 382.582,Z 362.905,A -85,B 0,C 180,E1 -12153.686,E2 -12153.686} C_VEL
LIN {X 0,Y 382.168,Z 368.696,A -85,B 0,C 180,E1 -12155.276,E2 -12155.276} C_VEL
LIN {X 0,Y 381.954,Z 373.118,A -85,B 0,C 180,E1 -12156.816,E2 -12156.816} C_VEL
LIN {X 0,Y 381.683,Z 376.732,A -85,B 0,C 180,E1 -12158.471,E2 -12158.471} C_VEL
LIN {X 0,Y 381.544,Z 378.467,A -85,B 0,C 180,E1 -12159.542,E2 -12159.542} C_VEL
LIN {X 0,Y 381.501,Z 379.787,A -85,B 0,C 180,E1 -12160.615,E2 -12160.615} C_VEL
LIN {X 0,Y 381.521,Z 381.115,A -85,B 0,C 180,E1 -12162.504,E2 -12162.504} C_VEL
LIN {X 0,Y 381.443,Z 381.272,A -85,B 0,C 180,E1 -12163.858,E2 -12163.858} C_VEL
LIN {X 0,Y 381.438,Z 380.942,A -85,B 0,C 180,E1 -12164.948,E2 -12164.948} C_VEL
LIN {X 0,Y 381.638,Z 379.471,A -85,B 0,C 180,E1 -12166.751,E2 -12166.751} C_VEL
LIN {X 0,Y 381.919,Z 376.379,A -85,B 0,C 180,E1 -12168.785,E2 -12168.785} C_VEL
LIN {X 0,Y 382.31,Z 372.663,A -85,B 0,C 180,E1 -12170.443,E2 -12170.443} C_VEL
LIN {X 0,Y 382.782,Z 367.729,A -85,B 0,C 180,E1 -12172.109,E2 -12172.109} C_VEL
LIN {X 0,Y 383.482,Z 361.419,A -85,B 0,C 180,E1 -12173.777,E2 -12173.777} C_VEL
LIN {X 0,Y 384.43,Z 353.471,A -85,B 0,C 180,E1 -12175.443,E2 -12175.443} C_VEL
LIN {X 0,Y 385.379,Z 345.089,A -85,B 0,C 180,E1 -12176.849,E2 -12176.849} C_VEL
LIN {X 0,Y 385.168,Z 341.002,A -85,B 0,C 180,E1 -12177.478,E2 -12177.478} C_VEL
LIN {X 0,Y 382.227,Z 331.34,A -85,B 0,C 180,E1 -12178.906,E2 -12178.906} C_VEL
LIN {X 0,Y 381.024,Z 325.322,A -85,B 0,C 180,E1 -12179.649,E2 -12179.649} C_VEL
LIN {X 0,Y 381.067,Z 322.032,A -85,B 0,C 180,E1 -12179.98,E2 -12179.98} C_VEL
LIN {X 0,Y 382.097,Z 310.765,A -85,B 0,C 180,E1 -12180.913,E2 -12180.913} C_VEL
LIN {X 0,Y 382.343,Z 306.618,A -85,B 0,C 180,E1 -12181.203,E2 -12181.203} C_VEL
LIN {X 0,Y 380.218,Z 295.477,A -85,B 0,C 180,E1 -12182.026,E2 -12182.026} C_VEL
LIN {X 0,Y 376.606,Z 282.521,A -85,B 0,C 180,E1 -12182.835,E2 -12182.835} C_VEL
LIN {X 0,Y 375.118,Z 277.439,A -85,B 0,C 180,E1 -12183.108,E2 -12183.108} C_VEL
LIN {X 0,Y 375.353,Z 272.895,A -85,B 0,C 180,E1 -12186.809,E2 -12186.809} C_VEL
LIN {X 0,Y 375.55,Z 269.226,A -85,B 0,C 180,E1 -12189.893,E2 -12189.893} C_VEL
LIN {X 0,Y 375.895,Z 264.733,A -85,B 0,C 180,E1 -12193.77,E2 -12193.77} C_VEL
LIN {X 0,Y 376.094,Z 261.403,A -85,B 0,C 180,E1 -12196.783,E2 -12196.783} C_VEL
LIN {X 0,Y 376.098,Z 257.991,A -85,B 0,C 180,E1 -12200.008,E2 -12200.008} C_VEL
LIN {X 0,Y 375.946,Z 256.658,A -85,B 0,C 180,E1 -12201.911,E2 -12201.911} C_VEL
LIN {X 0,Y 375.968,Z 256.657,A -85,B 0,C 180,E1 -12205.333,E2 -12205.333} C_VEL
LIN {X 0,Y 375.948,Z 256.659,A -85,B 0,C 180,E1 -12208.439,E2 -12208.439} C_VEL
LIN {X 0,Y 375.991,Z 256.651,A -85,B 0,C 180,E1 -12212.143,E2 -12212.143} C_VEL
LIN {X 0,Y 375.995,Z 256.651,A -85,B 0,C 180,E1 -12214.54,E2 -12214.54} C_VEL
LIN {X 0,Y 375.984,Z 256.653,A -85,B 0,C 180,E1 -12218.049,E2 -12218.049} C_VEL
LIN {X 0,Y 376.021,Z 256.646,A -85,B 0,C 180,E1 -12221.475,E2 -12221.475} C_VEL
LIN {X 0,Y 376.05,Z 256.642,A -85,B 0,C 180,E1 -12224.834,E2 -12224.834} C_VEL
LIN {X 0,Y 376.04,Z 256.645,A -85,B 0,C 180,E1 -12228.138,E2 -12228.138} C_VEL
LIN {X 0,Y 376.21,Z 256.623,A -85,B 0,C 180,E1 -12231.919,E2 -12231.919} C_VEL
LIN {X 0,Y 376.16,Z 256.631,A -85,B 0,C 180,E1 -12234.641,E2 -12234.641} C_VEL
LIN {X 0,Y 376.345,Z 256.607,A -85,B 0,C 180,E1 -12237.861,E2 -12237.861} C_VEL
LIN {X 0,Y 376.477,Z 256.588,A -85,B 0,C 180,E1 -12240.001,E2 -12240.001} C_VEL
LIN {X 0,Y 376.182,Z 256.628,A -85,B 0,C 180,E1 -12243.214,E2 -12243.214} C_VEL
LIN {X 0,Y 376.236,Z 256.621,A -85,B 0,C 180,E1 -12246.436,E2 -12246.436} C_VEL
LIN {X 0,Y 376.198,Z 256.625,A -85,B 0,C 180,E1 -12248.596,E2 -12248.596} C_VEL
LIN {X 0,Y 376.043,Z 256.643,A -85,B 0,C 180,E1 -12251.865,E2 -12251.865} C_VEL
LIN {X 0,Y 376.051,Z 256.645,A -85,B 0,C 180,E1 -12255.169,E2 -12255.169} C_VEL
LIN {X 0,Y 376.018,Z 256.652,A -85,B 0,C 180,E1 -12258.527,E2 -12258.527} C_VEL
LIN {X 0,Y 375.958,Z 256.659,A -85,B 0,C 180,E1 -12261.956,E2 -12261.956} C_VEL
LIN {X 0,Y 375.996,Z 256.654,A -85,B 0,C 180,E1 -12265.463,E2 -12265.463} C_VEL
LIN {X 0,Y 375.924,Z 256.663,A -85,B 0,C 180,E1 -12269.084,E2 -12269.084} C_VEL
LIN {X 0,Y 375.954,Z 256.657,A -85,B 0,C 180,E1 -12271.564,E2 -12271.564} C_VEL
LIN {X 0,Y 375.954,Z 256.657,A -85,B 0,C 180,E1 -12275.417,E2 -12275.417} C_VEL
LIN {X 0,Y 375.971,Z 256.654,A -85,B 0,C 180,E1 -12278.272,E2 -12278.272} C_VEL
LIN {X 0,Y 375.933,Z 256.658,A -85,B 0,C 180,E1 -12281.602,E2 -12281.602} C_VEL
LIN {X 0,Y 375.924,Z 256.651,A -85,B 0,C 180,E1 -12285.27,E2 -12285.27} C_VEL
LIN {X 0,Y 375.987,Z 256.924,A -85,B 0,C 180,E1 -12285.772,E2 -12285.772} C_VEL
LIN {X 0,Y 376.739,Z 261.445,A -85,B 0,C 180,E1 -12289.239,E2 -12289.239} C_VEL
LIN {X 0,Y 377.401,Z 265.421,A -85,B 0,C 180,E1 -12292.083,E2 -12292.083} C_VEL
LIN {X 0,Y 377.583,Z 269.435,A -85,B 0,C 180,E1 -12294.761,E2 -12294.761} C_VEL
LIN {X 0,Y 377.13,Z 274.523,A -85,B 0,C 180,E1 -12297.92,E2 -12297.92} C_VEL
LIN {X 0,Y 376.48,Z 280.283,A -85,B 0,C 180,E1 -12301.33,E2 -12301.33} C_VEL
LIN {X 0,Y 375.912,Z 286.929,A -85,B 0,C 180,E1 -12305.125,E2 -12305.125} C_VEL
LIN {X 0,Y 375.507,Z 293.195,A -85,B 0,C 180,E1 -12308.595,E2 -12308.595} C_VEL
LIN {X 0,Y 375.324,Z 295.795,A -85,B 0,C 180,E1 -12309.949,E2 -12309.949} C_VEL
LIN {X 0,Y 378.529,Z 309.069,A -85,B 0,C 180,E1 -12310.621,E2 -12310.621} C_VEL
LIN {X 0,Y 380.457,Z 320.044,A -85,B 0,C 180,E1 -12311.308,E2 -12311.308} C_VEL
LIN {X 0,Y 381.464,Z 329.849,A -85,B 0,C 180,E1 -12312.026,E2 -12312.026} C_VEL
LIN {X 0,Y 380.649,Z 339.813,A -85,B 0,C 180,E1 -12312.818,E2 -12312.818} C_VEL
LIN {X 0,Y 379.499,Z 350.492,A -85,B 0,C 180,E1 -12313.872,E2 -12313.872} C_VEL
LIN {X 0,Y 378.323,Z 361.216,A -85,B 0,C 180,E1 -12315.204,E2 -12315.204} C_VEL
LIN {X 0,Y 377.435,Z 369.919,A -85,B 0,C 180,E1 -12316.541,E2 -12316.541} C_VEL
LIN {X 0,Y 376.313,Z 378.442,A -85,B 0,C 180,E1 -12318.145,E2 -12318.145} C_VEL
LIN {X 0,Y 375.624,Z 385.284,A -85,B 0,C 180,E1 -12319.762,E2 -12319.762} C_VEL
LIN {X 0,Y 375.116,Z 390.783,A -85,B 0,C 180,E1 -12321.38,E2 -12321.38} C_VEL
LIN {X 0,Y 374.746,Z 395.113,A -85,B 0,C 180,E1 -12322.998,E2 -12322.998} C_VEL
LIN {X 0,Y 374.558,Z 398.388,A -85,B 0,C 180,E1 -12324.617,E2 -12324.617} C_VEL
LIN {X 0,Y 374.531,Z 400.026,A -85,B 0,C 180,E1 -12325.696,E2 -12325.696} C_VEL
LIN {X 0,Y 374.461,Z 401.264,A -85,B 0,C 180,E1 -12326.772,E2 -12326.772} C_VEL
LIN {X 0,Y 374.458,Z 402.083,A -85,B 0,C 180,E1 -12327.849,E2 -12327.849} C_VEL
LIN {X 0,Y 374.504,Z 402.486,A -85,B 0,C 180,E1 -12328.925,E2 -12328.925} C_VEL
LIN {X 0,Y 374.555,Z 402.506,A -85,B 0,C 180,E1 -12330,E2 -12330} C_VEL
LIN {X 0,Y 374.521,Z 402.137,A -85,B 0,C 180,E1 -12331.075,E2 -12331.075} C_VEL
LIN {X 0,Y 374.476,Z 401.362,A -85,B 0,C 180,E1 -12332.151,E2 -12332.151} C_VEL
LIN {X 0,Y 374.556,Z 398.531,A -85,B 0,C 180,E1 -12334.304,E2 -12334.304} C_VEL
LIN {X 0,Y 374.586,Z 394.931,A -85,B 0,C 180,E1 -12336.066,E2 -12336.066} C_VEL
LIN {X 0,Y 374.776,Z 390.916,A -85,B 0,C 180,E1 -12337.543,E2 -12337.543} C_VEL
LIN {X 0,Y 375.114,Z 385.366,A -85,B 0,C 180,E1 -12339.163,E2 -12339.163} C_VEL
LIN {X 0,Y 375.579,Z 378.422,A -85,B 0,C 180,E1 -12340.785,E2 -12340.785} C_VEL
LIN {X 0,Y 376.387,Z 369.724,A -85,B 0,C 180,E1 -12342.399,E2 -12342.399} C_VEL
LIN {X 0,Y 377.148,Z 360.788,A -85,B 0,C 180,E1 -12343.744,E2 -12343.744} C_VEL
LIN {X 0,Y 377.989,Z 349.76,A -85,B 0,C 180,E1 -12345.088,E2 -12345.088} C_VEL
LIN {X 0,Y 378.865,Z 338.581,A -85,B 0,C 180,E1 -12346.156,E2 -12346.156} C_VEL
LIN {X 0,Y 379.569,Z 328.032,A -85,B 0,C 180,E1 -12346.955,E2 -12346.955} C_VEL
LIN {X 0,Y 377.966,Z 314.995,A -85,B 0,C 180,E1 -12347.791,E2 -12347.791} C_VEL
LIN {X 0,Y 376.041,Z 302.256,A -85,B 0,C 180,E1 -12348.393,E2 -12348.393} C_VEL
LIN {X 0,Y 375.033,Z 295.951,A -85,B 0,C 180,E1 -12348.647,E2 -12348.647} C_VEL
LIN {X 0,Y 375.352,Z 289.564,A -85,B 0,C 180,E1 -12351.991,E2 -12351.991} C_VEL
LIN {X 0,Y 375.704,Z 283.001,A -85,B 0,C 180,E1 -12355.482,E2 -12355.482} C_VEL
LIN {X 0,Y 376.169,Z 276.416,A -85,B 0,C 180,E1 -12359.062,E2 -12359.062} C_VEL
LIN {X 0,Y 376.74,Z 269.829,A -85,B 0,C 180,E1 -12362.75,E2 -12362.75} C_VEL
LIN {X 0,Y 377.09,Z 264.298,A -85,B 0,C 180,E1 -12365.949,E2 -12365.949} C_VEL
LIN {X 0,Y 376.603,Z 260.337,A -85,B 0,C 180,E1 -12368.39,E2 -12368.39} C_VEL
LIN {X 0,Y 375.989,Z 256.653,A -85,B 0,C 180,E1 -12370.859,E2 -12370.859} C_VEL
LIN {X 0,Y 375.914,Z 256.661,A -85,B 0,C 180,E1 -12374.728,E2 -12374.728} C_VEL
LIN {X 0,Y 375.907,Z 256.659,A -85,B 0,C 180,E1 -12378.403,E2 -12378.403} C_VEL
LIN {X 0,Y 375.949,Z 256.652,A -85,B 0,C 180,E1 -12381.908,E2 -12381.908} C_VEL
LIN {X 0,Y 375.971,Z 256.651,A -85,B 0,C 180,E1 -12385.333,E2 -12385.333} C_VEL
LIN {X 0,Y 375.953,Z 256.656,A -85,B 0,C 180,E1 -12388.436,E2 -12388.436} C_VEL
LIN {X 0,Y 375.923,Z 256.658,A -85,B 0,C 180,E1 -12392.134,E2 -12392.134} C_VEL
LIN {X 0,Y 375.967,Z 256.651,A -85,B 0,C 180,E1 -12395.716,E2 -12395.716} C_VEL
LIN {X 0,Y 375.975,Z 256.65,A -85,B 0,C 180,E1 -12399.195,E2 -12399.195} C_VEL
LIN {X 0,Y 376.045,Z 256.644,A -85,B 0,C 180,E1 -12402.6,E2 -12402.6} C_VEL
LIN {X 0,Y 376.084,Z 256.64,A -85,B 0,C 180,E1 -12406.341,E2 -12406.341} C_VEL
LIN {X 0,Y 376.112,Z 256.637,A -85,B 0,C 180,E1 -12410.317,E2 -12410.317} C_VEL
LIN {X 0,Y 376.233,Z 256.619,A -85,B 0,C 180,E1 -12413.564,E2 -12413.564} C_VEL
LIN {X 0,Y 376.345,Z 256.608,A -85,B 0,C 180,E1 -12417.858,E2 -12417.858} C_VEL
LIN {X 0,Y 376.482,Z 256.591,A -85,B 0,C 180,E1 -12419.999,E2 -12419.999} C_VEL
LIN {X 0,Y 376.183,Z 256.625,A -85,B 0,C 180,E1 -12423.212,E2 -12423.212} C_VEL
LIN {X 0,Y 376.225,Z 256.618,A -85,B 0,C 180,E1 -12426.644,E2 -12426.644} C_VEL
LIN {X 0,Y 376.196,Z 256.622,A -85,B 0,C 180,E1 -12428.594,E2 -12428.594} C_VEL
LIN {X 0,Y 376.041,Z 256.645,A -85,B 0,C 180,E1 -12431.862,E2 -12431.862} C_VEL
LIN {X 0,Y 376.048,Z 256.643,A -85,B 0,C 180,E1 -12435.166,E2 -12435.166} C_VEL
LIN {X 0,Y 375.998,Z 256.647,A -85,B 0,C 180,E1 -12438.526,E2 -12438.526} C_VEL
LIN {X 0,Y 375.952,Z 256.653,A -85,B 0,C 180,E1 -12441.953,E2 -12441.953} C_VEL
LIN {X 0,Y 375.996,Z 256.651,A -85,B 0,C 180,E1 -12445.46,E2 -12445.46} C_VEL
LIN {X 0,Y 375.965,Z 256.654,A -85,B 0,C 180,E1 -12449.078,E2 -12449.078} C_VEL
LIN {X 0,Y 375.938,Z 256.657,A -85,B 0,C 180,E1 -12452.828,E2 -12452.828} C_VEL
LIN {X 0,Y 375.947,Z 256.655,A -85,B 0,C 180,E1 -12455.415,E2 -12455.415} C_VEL
LIN {X 0,Y 375.966,Z 256.65,A -85,B 0,C 180,E1 -12458.271,E2 -12458.271} C_VEL
LIN {X 0,Y 375.978,Z 256.649,A -85,B 0,C 180,E1 -12461.61,E2 -12461.61} C_VEL
LIN {X 0,Y 375.958,Z 256.653,A -85,B 0,C 180,E1 -12465.261,E2 -12465.261} C_VEL
LIN {X 0,Y 375.929,Z 256.657,A -85,B 0,C 180,E1 -12469.133,E2 -12469.133} C_VEL
LIN {X 0,Y 375.954,Z 256.652,A -85,B 0,C 180,E1 -12471.911,E2 -12471.911} C_VEL
LIN {X 0,Y 375.968,Z 256.65,A -85,B 0,C 180,E1 -12475.332,E2 -12475.332} C_VEL
LIN {X 0,Y 375.945,Z 256.658,A -85,B 0,C 180,E1 -12478.438,E2 -12478.438} C_VEL
LIN {X 0,Y 375.97,Z 256.653,A -85,B 0,C 180,E1 -12482.14,E2 -12482.14} C_VEL
LIN {X 0,Y 375.951,Z 256.656,A -85,B 0,C 180,E1 -12484.536,E2 -12484.536} C_VEL
LIN {X 0,Y 375.857,Z 256.665,A -85,B 0,C 180,E1 -12486.88,E2 -12486.88} C_VEL
LIN {X 0,Y 375.71,Z 256.745,A -85,B 0,C 180,E1 -12488.319,E2 -12488.319} C_VEL
LIN {X 0,Y 375.634,Z 260.507,A -85,B 0,C 180,E1 -12491.454,E2 -12491.454} C_VEL
LIN {X 0,Y 375.435,Z 264.657,A -85,B 0,C 180,E1 -12494.807,E2 -12494.807} C_VEL
LIN {X 0,Y 375.441,Z 267.429,A -85,B 0,C 180,E1 -12497.019,E2 -12497.019} C_VEL
LIN {X 0,Y 375.216,Z 273.042,A -85,B 0,C 180,E1 -12501.382,E2 -12501.382} C_VEL
LIN {X 0,Y 375.156,Z 276.58,A -85,B 0,C 180,E1 -12504.086,E2 -12504.086} C_VEL
LIN {X 0,Y 375.093,Z 277.075,A -85,B 0,C 180,E1 -12504.456,E2 -12504.456} C_VEL
LIN {X 0,Y 378.089,Z 291.915,A -85,B 0,C 180,E1 -12505.152,E2 -12505.152} C_VEL
LIN {X 0,Y 380.071,Z 303.92,A -85,B 0,C 180,E1 -12505.891,E2 -12505.891} C_VEL
LIN {X 0,Y 379.528,Z 315.024,A -85,B 0,C 180,E1 -12506.683,E2 -12506.683} C_VEL
LIN {X 0,Y 378.635,Z 326.605,A -85,B 0,C 180,E1 -12507.74,E2 -12507.74} C_VEL
LIN {X 0,Y 377.862,Z 337.002,A -85,B 0,C 180,E1 -12508.934,E2 -12508.934} C_VEL
LIN {X 0,Y 376.942,Z 346.421,A -85,B 0,C 180,E1 -12510.267,E2 -12510.267} C_VEL
LIN {X 0,Y 376.121,Z 355.479,A -85,B 0,C 180,E1 -12511.874,E2 -12511.874} C_VEL
LIN {X 0,Y 375.583,Z 362.773,A -85,B 0,C 180,E1 -12513.486,E2 -12513.486} C_VEL
LIN {X 0,Y 375.132,Z 367.734,A -85,B 0,C 180,E1 -12514.836,E2 -12514.836} C_VEL
LIN {X 0,Y 374.909,Z 372.747,A -85,B 0,C 180,E1 -12516.537,E2 -12516.537} C_VEL
LIN {X 0,Y 374.661,Z 376.242,A -85,B 0,C 180,E1 -12518.087,E2 -12518.087} C_VEL
LIN {X 0,Y 374.431,Z 378.928,A -85,B 0,C 180,E1 -12519.725,E2 -12519.725} C_VEL
LIN {X 0,Y 374.408,Z 380.189,A -85,B 0,C 180,E1 -12520.819,E2 -12520.819} C_VEL
LIN {X 0,Y 374.423,Z 381.326,A -85,B 0,C 180,E1 -12522.573,E2 -12522.573} C_VEL
LIN {X 0,Y 374.353,Z 381.446,A -85,B 0,C 180,E1 -12524.126,E2 -12524.126} C_VEL
LIN {X 0,Y 374.371,Z 381.058,A -85,B 0,C 180,E1 -12525.237,E2 -12525.237} C_VEL
LIN {X 0,Y 374.573,Z 379.66,A -85,B 0,C 180,E1 -12526.89,E2 -12526.89} C_VEL
LIN {X 0,Y 374.926,Z 376.193,A -85,B 0,C 180,E1 -12529.149,E2 -12529.149} C_VEL
LIN {X 0,Y 375.331,Z 372.346,A -85,B 0,C 180,E1 -12530.84,E2 -12530.84} C_VEL
LIN {X 0,Y 375.886,Z 367.273,A -85,B 0,C 180,E1 -12532.537,E2 -12532.537} C_VEL
LIN {X 0,Y 376.658,Z 360.812,A -85,B 0,C 180,E1 -12534.235,E2 -12534.235} C_VEL
LIN {X 0,Y 377.693,Z 352.603,A -85,B 0,C 180,E1 -12535.93,E2 -12535.93} C_VEL
LIN {X 0,Y 378.744,Z 343.637,A -85,B 0,C 180,E1 -12537.418,E2 -12537.418} C_VEL
LIN {X 0,Y 379.892,Z 333.68,A -85,B 0,C 180,E1 -12538.75,E2 -12538.75} C_VEL
LIN {X 0,Y 380.964,Z 323.039,A -85,B 0,C 180,E1 -12539.886,E2 -12539.886} C_VEL
LIN {X 0,Y 381.067,Z 322.032,A -85,B 0,C 180,E1 -12539.98,E2 -12539.98} C_VEL
LIN {X 0,Y 380.876,Z 317.055,A -85,B 0,C 180,E1 -12540.462,E2 -12540.462} C_VEL
LIN {X 0,Y 379.605,Z 312.217,A -85,B 0,C 180,E1 -12540.951,E2 -12540.951} C_VEL
LIN {X 0,Y 374.398,Z 299.286,A -85,B 0,C 180,E1 -12542.189,E2 -12542.189} C_VEL
LIN {X 0,Y 373.323,Z 295.803,A -85,B 0,C 180,E1 -12542.457,E2 -12542.457} C_VEL
LIN {X 0,Y 369.681,Z 282.961,A -85,B 0,C 180,E1 -12543.292,E2 -12543.292} C_VEL
LIN {X 0,Y 368.1,Z 277.641,A -85,B 0,C 180,E1 -12543.586,E2 -12543.586} C_VEL
LIN {X 0,Y 368.362,Z 272.791,A -85,B 0,C 180,E1 -12547.627,E2 -12547.627} C_VEL
LIN {X 0,Y 368.551,Z 269.544,A -85,B 0,C 180,E1 -12550.416,E2 -12550.416} C_VEL
LIN {X 0,Y 368.848,Z 265.918,A -85,B 0,C 180,E1 -12553.613,E2 -12553.613} C_VEL
LIN {X 0,Y 369.074,Z 262.523,A -85,B 0,C 180,E1 -12556.726,E2 -12556.726} C_VEL
LIN {X 0,Y 369.096,Z 259.47,A -85,B 0,C 180,E1 -12559.657,E2 -12559.657} C_VEL
LIN {X 0,Y 368.915,Z 257.793,A -85,B 0,C 180,E1 -12561.357,E2 -12561.357} C_VEL
LIN {X 0,Y 368.905,Z 257.535,A -85,B 0,C 180,E1 -12563.804,E2 -12563.804} C_VEL
LIN {X 0,Y 368.885,Z 257.54,A -85,B 0,C 180,E1 -12566.958,E2 -12566.958} C_VEL
LIN {X 0,Y 368.911,Z 257.536,A -85,B 0,C 180,E1 -12570.311,E2 -12570.311} C_VEL
LIN {X 0,Y 368.97,Z 257.527,A -85,B 0,C 180,E1 -12573.536,E2 -12573.536} C_VEL
LIN {X 0,Y 368.969,Z 257.525,A -85,B 0,C 180,E1 -12576.423,E2 -12576.423} C_VEL
LIN {X 0,Y 368.945,Z 257.527,A -85,B 0,C 180,E1 -12579.949,E2 -12579.949} C_VEL
LIN {X 0,Y 368.968,Z 257.524,A -85,B 0,C 180,E1 -12583.4,E2 -12583.4} C_VEL
LIN {X 0,Y 369.047,Z 257.516,A -85,B 0,C 180,E1 -12586.791,E2 -12586.791} C_VEL
LIN {X 0,Y 369.058,Z 257.516,A -85,B 0,C 180,E1 -12590.133,E2 -12590.133} C_VEL
LIN {X 0,Y 369.19,Z 257.496,A -85,B 0,C 180,E1 -12593.443,E2 -12593.443} C_VEL
LIN {X 0,Y 369.31,Z 257.483,A -85,B 0,C 180,E1 -12597.82,E2 -12597.82} C_VEL
LIN {X 0,Y 369.446,Z 257.464,A -85,B 0,C 180,E1 -12600.001,E2 -12600.001} C_VEL
LIN {X 0,Y 369.31,Z 257.484,A -85,B 0,C 180,E1 -12602.182,E2 -12602.182} C_VEL
LIN {X 0,Y 369.198,Z 257.498,A -85,B 0,C 180,E1 -12606.56,E2 -12606.56} C_VEL
LIN {X 0,Y 369.13,Z 257.505,A -85,B 0,C 180,E1 -12608.762,E2 -12608.762} C_VEL
LIN {X 0,Y 368.998,Z 257.521,A -85,B 0,C 180,E1 -12612.095,E2 -12612.095} C_VEL
LIN {X 0,Y 368.991,Z 257.525,A -85,B 0,C 180,E1 -12615.466,E2 -12615.466} C_VEL
LIN {X 0,Y 368.977,Z 257.527,A -85,B 0,C 180,E1 -12618.894,E2 -12618.894} C_VEL
LIN {X 0,Y 368.927,Z 257.534,A -85,B 0,C 180,E1 -12622.397,E2 -12622.397} C_VEL
LIN {X 0,Y 368.966,Z 257.531,A -85,B 0,C 180,E1 -12625.984,E2 -12625.984} C_VEL
LIN {X 0,Y 368.896,Z 257.538,A -85,B 0,C 180,E1 -12629.693,E2 -12629.693} C_VEL
LIN {X 0,Y 368.894,Z 257.537,A -85,B 0,C 180,E1 -12633.54,E2 -12633.54} C_VEL
LIN {X 0,Y 368.899,Z 257.536,A -85,B 0,C 180,E1 -12636.857,E2 -12636.857} C_VEL
LIN {X 0,Y 368.909,Z 257.528,A -85,B 0,C 180,E1 -12640.372,E2 -12640.372} C_VEL
LIN {X 0,Y 368.881,Z 257.535,A -85,B 0,C 180,E1 -12643.617,E2 -12643.617} C_VEL
LIN {X 0,Y 368.905,Z 257.635,A -85,B 0,C 180,E1 -12645.181,E2 -12645.181} C_VEL
LIN {X 0,Y 369.584,Z 261.525,A -85,B 0,C 180,E1 -12648.276,E2 -12648.276} C_VEL
LIN {X 0,Y 370.229,Z 265.472,A -85,B 0,C 180,E1 -12651.214,E2 -12651.214} C_VEL
LIN {X 0,Y 370.61,Z 269.466,A -85,B 0,C 180,E1 -12653.996,E2 -12653.996} C_VEL
LIN {X 0,Y 370.313,Z 273.554,A -85,B 0,C 180,E1 -12656.623,E2 -12656.623} C_VEL
LIN {X 0,Y 369.757,Z 278.625,A -85,B 0,C 180,E1 -12659.757,E2 -12659.757} C_VEL
LIN {X 0,Y 369.098,Z 284.966,A -85,B 0,C 180,E1 -12663.501,E2 -12663.501} C_VEL
LIN {X 0,Y 368.649,Z 291.052,A -85,B 0,C 180,E1 -12666.995,E2 -12666.995} C_VEL
LIN {X 0,Y 368.337,Z 295.684,A -85,B 0,C 180,E1 -12669.476,E2 -12669.476} C_VEL
LIN {X 0,Y 371.614,Z 309.063,A -85,B 0,C 180,E1 -12670.18,E2 -12670.18} C_VEL
LIN {X 0,Y 373.732,Z 320.905,A -85,B 0,C 180,E1 -12670.959,E2 -12670.959} C_VEL
LIN {X 0,Y 374.709,Z 330.479,A -85,B 0,C 180,E1 -12671.69,E2 -12671.69} C_VEL
LIN {X 0,Y 373.912,Z 340.288,A -85,B 0,C 180,E1 -12672.499,E2 -12672.499} C_VEL
LIN {X 0,Y 372.575,Z 351.993,A -85,B 0,C 180,E1 -12673.705,E2 -12673.705} C_VEL
LIN {X 0,Y 371.405,Z 362.004,A -85,B 0,C 180,E1 -12675,E2 -12675} C_VEL
LIN {X 0,Y 370.51,Z 370.091,A -85,B 0,C 180,E1 -12676.285,E2 -12676.285} C_VEL
LIN {X 0,Y 369.353,Z 378.522,A -85,B 0,C 180,E1 -12677.919,E2 -12677.919} C_VEL
LIN {X 0,Y 368.609,Z 385.313,A -85,B 0,C 180,E1 -12679.565,E2 -12679.565} C_VEL
LIN {X 0,Y 368.068,Z 390.766,A -85,B 0,C 180,E1 -12681.214,E2 -12681.214} C_VEL
LIN {X 0,Y 367.685,Z 395.051,A -85,B 0,C 180,E1 -12682.863,E2 -12682.863} C_VEL
LIN {X 0,Y 367.472,Z 398.285,A -85,B 0,C 180,E1 -12684.513,E2 -12684.513} C_VEL
LIN {X 0,Y 367.439,Z 399.903,A -85,B 0,C 180,E1 -12685.612,E2 -12685.612} C_VEL
LIN {X 0,Y 367.379,Z 401.123,A -85,B 0,C 180,E1 -12686.71,E2 -12686.71} C_VEL
LIN {X 0,Y 367.359,Z 401.908,A -85,B 0,C 180,E1 -12687.807,E2 -12687.807} C_VEL
LIN {X 0,Y 367.404,Z 402.294,A -85,B 0,C 180,E1 -12688.904,E2 -12688.904} C_VEL
LIN {X 0,Y 367.458,Z 402.297,A -85,B 0,C 180,E1 -12690,E2 -12690} C_VEL
LIN {X 0,Y 367.422,Z 401.912,A -85,B 0,C 180,E1 -12691.096,E2 -12691.096} C_VEL
LIN {X 0,Y 367.377,Z 401.103,A -85,B 0,C 180,E1 -12692.193,E2 -12692.193} C_VEL
LIN {X 0,Y 367.383,Z 399.871,A -85,B 0,C 180,E1 -12693.29,E2 -12693.29} C_VEL
LIN {X 0,Y 367.45,Z 397.249,A -85,B 0,C 180,E1 -12694.937,E2 -12694.937} C_VEL
LIN {X 0,Y 367.567,Z 393.597,A -85,B 0,C 180,E1 -12696.587,E2 -12696.587} C_VEL
LIN {X 0,Y 367.81,Z 388.817,A -85,B 0,C 180,E1 -12698.239,E2 -12698.239} C_VEL
LIN {X 0,Y 368.328,Z 381.638,A -85,B 0,C 180,E1 -12700.166,E2 -12700.166} C_VEL
LIN {X 0,Y 368.968,Z 373.794,A -85,B 0,C 180,E1 -12701.815,E2 -12701.815} C_VEL
LIN {X 0,Y 369.661,Z 365.768,A -85,B 0,C 180,E1 -12703.188,E2 -12703.188} C_VEL
LIN {X 0,Y 370.488,Z 356.447,A -85,B 0,C 180,E1 -12704.495,E2 -12704.495} C_VEL
LIN {X 0,Y 371.363,Z 345.048,A -85,B 0,C 180,E1 -12705.786,E2 -12705.786} C_VEL
LIN {X 0,Y 372.324,Z 334.389,A -85,B 0,C 180,E1 -12706.73,E2 -12706.73} C_VEL
LIN {X 0,Y 372.539,Z 327.886,A -85,B 0,C 180,E1 -12707.214,E2 -12707.214} C_VEL
LIN {X 0,Y 370.947,Z 314.956,A -85,B 0,C 180,E1 -12708.063,E2 -12708.063} C_VEL
LIN {X 0,Y 368.945,Z 301.939,A -85,B 0,C 180,E1 -12708.694,E2 -12708.694} C_VEL
LIN {X 0,Y 367.969,Z 295.774,A -85,B 0,C 180,E1 -12708.946,E2 -12708.946} C_VEL
LIN {X 0,Y 368.307,Z 289.257,A -85,B 0,C 180,E1 -12712.435,E2 -12712.435} C_VEL
LIN {X 0,Y 368.718,Z 282.702,A -85,B 0,C 180,E1 -12716.001,E2 -12716.001} C_VEL
LIN {X 0,Y 369.217,Z 276.134,A -85,B 0,C 180,E1 -12719.663,E2 -12719.663} C_VEL
LIN {X 0,Y 369.779,Z 269.533,A -85,B 0,C 180,E1 -12723.447,E2 -12723.447} C_VEL
LIN {X 0,Y 370.046,Z 265.118,A -85,B 0,C 180,E1 -12726.068,E2 -12726.068} C_VEL
LIN {X 0,Y 369.496,Z 260.852,A -85,B 0,C 180,E1 -12728.753,E2 -12728.753} C_VEL
LIN {X 0,Y 368.931,Z 257.533,A -85,B 0,C 180,E1 -12730.995,E2 -12730.995} C_VEL
LIN {X 0,Y 368.865,Z 257.54,A -85,B 0,C 180,E1 -12734.825,E2 -12734.825} C_VEL
LIN {X 0,Y 368.854,Z 257.537,A -85,B 0,C 180,E1 -12738.172,E2 -12738.172} C_VEL
LIN {X 0,Y 368.873,Z 257.535,A -85,B 0,C 180,E1 -12741.365,E2 -12741.365} C_VEL
LIN {X 0,Y 368.927,Z 257.529,A -85,B 0,C 180,E1 -12745.144,E2 -12745.144} C_VEL
LIN {X 0,Y 368.91,Z 257.532,A -85,B 0,C 180,E1 -12749.043,E2 -12749.043} C_VEL
LIN {X 0,Y 368.908,Z 257.53,A -85,B 0,C 180,E1 -12751.557,E2 -12751.557} C_VEL
LIN {X 0,Y 368.921,Z 257.528,A -85,B 0,C 180,E1 -12755.221,E2 -12755.221} C_VEL
LIN {X 0,Y 368.915,Z 257.53,A -85,B 0,C 180,E1 -12758.979,E2 -12758.979} C_VEL
LIN {X 0,Y 368.986,Z 257.525,A -85,B 0,C 180,E1 -12762.256,E2 -12762.256} C_VEL
LIN {X 0,Y 369.031,Z 257.519,A -85,B 0,C 180,E1 -12766.227,E2 -12766.227} C_VEL
LIN {X 0,Y 369.061,Z 257.515,A -85,B 0,C 180,E1 -12770.13,E2 -12770.13} C_VEL
LIN {X 0,Y 369.193,Z 257.495,A -85,B 0,C 180,E1 -12773.44,E2 -12773.44} C_VEL
LIN {X 0,Y 369.31,Z 257.484,A -85,B 0,C 180,E1 -12777.818,E2 -12777.818} C_VEL
LIN {X 0,Y 369.452,Z 257.467,A -85,B 0,C 180,E1 -12779.999,E2 -12779.999} C_VEL
LIN {X 0,Y 369.311,Z 257.483,A -85,B 0,C 180,E1 -12782.18,E2 -12782.18} C_VEL
LIN {X 0,Y 369.194,Z 257.494,A -85,B 0,C 180,E1 -12786.632,E2 -12786.632} C_VEL
LIN {X 0,Y 369.129,Z 257.502,A -85,B 0,C 180,E1 -12788.76,E2 -12788.76} C_VEL
LIN {X 0,Y 368.996,Z 257.52,A -85,B 0,C 180,E1 -12792.092,E2 -12792.092} C_VEL
LIN {X 0,Y 368.987,Z 257.524,A -85,B 0,C 180,E1 -12795.464,E2 -12795.464} C_VEL
LIN {X 0,Y 368.948,Z 257.526,A -85,B 0,C 180,E1 -12798.893,E2 -12798.893} C_VEL
LIN {X 0,Y 368.921,Z 257.528,A -85,B 0,C 180,E1 -12802.394,E2 -12802.394} C_VEL
LIN {X 0,Y 368.989,Z 257.52,A -85,B 0,C 180,E1 -12805.979,E2 -12805.979} C_VEL
LIN {X 0,Y 368.956,Z 257.526,A -85,B 0,C 180,E1 -12808.812,E2 -12808.812} C_VEL
LIN {X 0,Y 368.888,Z 257.532,A -85,B 0,C 180,E1 -12812.237,E2 -12812.237} C_VEL
LIN {X 0,Y 368.918,Z 257.533,A -85,B 0,C 180,E1 -12815.001,E2 -12815.001} C_VEL
LIN {X 0,Y 368.902,Z 257.533,A -85,B 0,C 180,E1 -12818.641,E2 -12818.641} C_VEL
LIN {X 0,Y 368.93,Z 257.526,A -85,B 0,C 180,E1 -12822.019,E2 -12822.019} C_VEL
LIN {X 0,Y 368.913,Z 257.531,A -85,B 0,C 180,E1 -12825.182,E2 -12825.182} C_VEL
LIN {X 0,Y 368.871,Z 257.534,A -85,B 0,C 180,E1 -12828.177,E2 -12828.177} C_VEL
LIN {X 0,Y 368.898,Z 257.531,A -85,B 0,C 180,E1 -12831.359,E2 -12831.359} C_VEL
LIN {X 0,Y 368.925,Z 257.528,A -85,B 0,C 180,E1 -12835.146,E2 -12835.146} C_VEL
LIN {X 0,Y 368.918,Z 257.529,A -85,B 0,C 180,E1 -12839.046,E2 -12839.046} C_VEL
LIN {X 0,Y 368.95,Z 257.524,A -85,B 0,C 180,E1 -12841.562,E2 -12841.562} C_VEL
LIN {X 0,Y 368.949,Z 257.527,A -85,B 0,C 180,E1 -12844.017,E2 -12844.017} C_VEL
LIN {X 0,Y 368.876,Z 257.538,A -85,B 0,C 180,E1 -12846.416,E2 -12846.416} C_VEL
LIN {X 0,Y 368.676,Z 257.632,A -85,B 0,C 180,E1 -12848.325,E2 -12848.325} C_VEL
LIN {X 0,Y 368.602,Z 260.914,A -85,B 0,C 180,E1 -12851.087,E2 -12851.087} C_VEL
LIN {X 0,Y 368.409,Z 265.05,A -85,B 0,C 180,E1 -12854.51,E2 -12854.51} C_VEL
LIN {X 0,Y 368.291,Z 269.241,A -85,B 0,C 180,E1 -12857.883,E2 -12857.883} C_VEL
LIN {X 0,Y 368.139,Z 273.467,A -85,B 0,C 180,E1 -12861.215,E2 -12861.215} C_VEL
LIN {X 0,Y 368.08,Z 277.3,A -85,B 0,C 180,E1 -12864.178,E2 -12864.178} C_VEL
LIN {X 0,Y 370.856,Z 290.866,A -85,B 0,C 180,E1 -12864.801,E2 -12864.801} C_VEL
LIN {X 0,Y 372.757,Z 302.944,A -85,B 0,C 180,E1 -12865.539,E2 -12865.539} C_VEL
LIN {X 0,Y 373.176,Z 306.814,A -85,B 0,C 180,E1 -12865.815,E2 -12865.815} C_VEL
LIN {X 0,Y 372.36,Z 318.949,A -85,B 0,C 180,E1 -12866.754,E2 -12866.754} C_VEL
LIN {X 0,Y 371.419,Z 329.809,A -85,B 0,C 180,E1 -12867.831,E2 -12867.831} C_VEL
LIN {X 0,Y 370.738,Z 338.628,A -85,B 0,C 180,E1 -12868.914,E2 -12868.914} C_VEL
LIN {X 0,Y 369.861,Z 347.731,A -85,B 0,C 180,E1 -12870.272,E2 -12870.272} C_VEL
LIN {X 0,Y 368.998,Z 356.608,A -85,B 0,C 180,E1 -12871.91,E2 -12871.91} C_VEL
LIN {X 0,Y 368.453,Z 363.733,A -85,B 0,C 180,E1 -12873.554,E2 -12873.554} C_VEL
LIN {X 0,Y 368.039,Z 368.558,A -85,B 0,C 180,E1 -12874.929,E2 -12874.929} C_VEL
LIN {X 0,Y 367.828,Z 373.231,A -85,B 0,C 180,E1 -12876.583,E2 -12876.583} C_VEL
LIN {X 0,Y 367.546,Z 376.816,A -85,B 0,C 180,E1 -12878.245,E2 -12878.245} C_VEL
LIN {X 0,Y 367.321,Z 379.384,A -85,B 0,C 180,E1 -12879.915,E2 -12879.915} C_VEL
LIN {X 0,Y 367.329,Z 380.575,A -85,B 0,C 180,E1 -12881.03,E2 -12881.03} C_VEL
LIN {X 0,Y 367.339,Z 381.54,A -85,B 0,C 180,E1 -12882.655,E2 -12882.655} C_VEL
LIN {X 0,Y 367.251,Z 381.621,A -85,B 0,C 180,E1 -12884.405,E2 -12884.405} C_VEL
LIN {X 0,Y 367.325,Z 381.141,A -85,B 0,C 180,E1 -12885.537,E2 -12885.537} C_VEL
LIN {X 0,Y 367.495,Z 379.863,A -85,B 0,C 180,E1 -12887.026,E2 -12887.026} C_VEL
LIN {X 0,Y 367.795,Z 377.111,A -85,B 0,C 180,E1 -12888.956,E2 -12888.956} C_VEL
LIN {X 0,Y 368.248,Z 373.321,A -85,B 0,C 180,E1 -12890.751,E2 -12890.751} C_VEL
LIN {X 0,Y 368.782,Z 368.705,A -85,B 0,C 180,E1 -12892.404,E2 -12892.404} C_VEL
LIN {X 0,Y 369.649,Z 361.748,A -85,B 0,C 180,E1 -12894.33,E2 -12894.33} C_VEL
LIN {X 0,Y 370.605,Z 354.774,A -85,B 0,C 180,E1 -12895.859,E2 -12895.859} C_VEL
LIN {X 0,Y 371.732,Z 345.808,A -85,B 0,C 180,E1 -12897.446,E2 -12897.446} C_VEL
LIN {X 0,Y 372.927,Z 335.711,A -85,B 0,C 180,E1 -12898.875,E2 -12898.875} C_VEL
LIN {X 0,Y 374.157,Z 324.786,A -85,B 0,C 180,E1 -12900.11,E2 -12900.11} C_VEL
LIN {X 0,Y 375.154,Z 314.814,A -85,B 0,C 180,E1 -12901.008,E2 -12901.008} C_VEL
LIN {X 0,Y 375.638,Z 307.741,A -85,B 0,C 180,E1 -12901.539,E2 -12901.539} C_VEL
LIN {X 0,Y 373.323,Z 295.803,A -85,B 0,C 180,E1 -12902.457,E2 -12902.457} C_VEL
LIN {X 0,Y 371.895,Z 292.572,A -85,B 0,C 180,E1 -12902.73,E2 -12902.73} C_VEL
LIN {X 0,Y 368.01,Z 288.108,A -85,B 0,C 180,E1 -12903.211,E2 -12903.211} C_VEL
LIN {X 0,Y 363.044,Z 282.737,A -85,B 0,C 180,E1 -12903.768,E2 -12903.768} C_VEL
LIN {X 0,Y 361.812,Z 280.58,A -85,B 0,C 180,E1 -12903.932,E2 -12903.932} C_VEL
LIN {X 0,Y 361.065,Z 277.833,A -85,B 0,C 180,E1 -12904.115,E2 -12904.115} C_VEL
LIN {X 0,Y 361.283,Z 274.286,A -85,B 0,C 180,E1 -12907.104,E2 -12907.104} C_VEL
LIN {X 0,Y 361.516,Z 270.172,A -85,B 0,C 180,E1 -12910.699,E2 -12910.699} C_VEL
LIN {X 0,Y 361.872,Z 266.123,A -85,B 0,C 180,E1 -12914.359,E2 -12914.359} C_VEL
LIN {X 0,Y 362.091,Z 262.775,A -85,B 0,C 180,E1 -12917.522,E2 -12917.522} C_VEL
LIN {X 0,Y 362.038,Z 260.096,A -85,B 0,C 180,E1 -12920.165,E2 -12920.165} C_VEL
LIN {X 0,Y 361.894,Z 258.738,A -85,B 0,C 180,E1 -12921.581,E2 -12921.581} C_VEL
LIN {X 0,Y 361.854,Z 258.412,A -85,B 0,C 180,E1 -12922.982,E2 -12922.982} C_VEL
LIN {X 0,Y 361.847,Z 258.417,A -85,B 0,C 180,E1 -12926.631,E2 -12926.631} C_VEL
LIN {X 0,Y 361.865,Z 258.411,A -85,B 0,C 180,E1 -12929.673,E2 -12929.673} C_VEL
LIN {X 0,Y 361.943,Z 258.402,A -85,B 0,C 180,E1 -12933.476,E2 -12933.476} C_VEL
LIN {X 0,Y 361.898,Z 258.403,A -85,B 0,C 180,E1 -12937.147,E2 -12937.147} C_VEL
LIN {X 0,Y 361.922,Z 258.404,A -85,B 0,C 180,E1 -12940.726,E2 -12940.726} C_VEL
LIN {X 0,Y 361.937,Z 258.401,A -85,B 0,C 180,E1 -12944.227,E2 -12944.227} C_VEL
LIN {X 0,Y 361.988,Z 258.393,A -85,B 0,C 180,E1 -12946.529,E2 -12946.529} C_VEL
LIN {X 0,Y 362.022,Z 258.391,A -85,B 0,C 180,E1 -12949.939,E2 -12949.939} C_VEL
LIN {X 0,Y 362.152,Z 258.373,A -85,B 0,C 180,E1 -12953.315,E2 -12953.315} C_VEL
LIN {X 0,Y 362.274,Z 258.359,A -85,B 0,C 180,E1 -12957.778,E2 -12957.778} C_VEL
LIN {X 0,Y 362.416,Z 258.34,A -85,B 0,C 180,E1 -12960.001,E2 -12960.001} C_VEL
LIN {X 0,Y 362.274,Z 258.361,A -85,B 0,C 180,E1 -12962.225,E2 -12962.225} C_VEL
LIN {X 0,Y 362.162,Z 258.375,A -85,B 0,C 180,E1 -12966.688,E2 -12966.688} C_VEL
LIN {X 0,Y 362.067,Z 258.385,A -85,B 0,C 180,E1 -12968.935,E2 -12968.935} C_VEL
LIN {X 0,Y 361.954,Z 258.4,A -85,B 0,C 180,E1 -12972.334,E2 -12972.334} C_VEL
LIN {X 0,Y 361.956,Z 258.4,A -85,B 0,C 180,E1 -12974.622,E2 -12974.622} C_VEL
LIN {X 0,Y 361.954,Z 258.402,A -85,B 0,C 180,E1 -12978.101,E2 -12978.101} C_VEL
LIN {X 0,Y 361.887,Z 258.414,A -85,B 0,C 180,E1 -12981.654,E2 -12981.654} C_VEL
LIN {X 0,Y 361.911,Z 258.409,A -85,B 0,C 180,E1 -12985.293,E2 -12985.293} C_VEL
LIN {X 0,Y 361.871,Z 258.414,A -85,B 0,C 180,E1 -12989.081,E2 -12989.081} C_VEL
LIN {X 0,Y 361.845,Z 258.414,A -85,B 0,C 180,E1 -12992.946,E2 -12992.946} C_VEL
LIN {X 0,Y 361.865,Z 258.411,A -85,B 0,C 180,E1 -12995.638,E2 -12995.638} C_VEL
LIN {X 0,Y 361.867,Z 258.409,A -85,B 0,C 180,E1 -12999.028,E2 -12999.028} C_VEL
LIN {X 0,Y 361.835,Z 258.412,A -85,B 0,C 180,E1 -13002.83,E2 -13002.83} C_VEL
LIN {X 0,Y 361.839,Z 258.514,A -85,B 0,C 180,E1 -13004.7,E2 -13004.7} C_VEL
LIN {X 0,Y 362.449,Z 261.867,A -85,B 0,C 180,E1 -13007.464,E2 -13007.464} C_VEL
LIN {X 0,Y 363.118,Z 266.112,A -85,B 0,C 180,E1 -13010.732,E2 -13010.732} C_VEL
LIN {X 0,Y 363.547,Z 269.502,A -85,B 0,C 180,E1 -13013.182,E2 -13013.182} C_VEL
LIN {X 0,Y 363.53,Z 272.521,A -85,B 0,C 180,E1 -13015.229,E2 -13015.229} C_VEL
LIN {X 0,Y 362.964,Z 277.606,A -85,B 0,C 180,E1 -13018.481,E2 -13018.481} C_VEL
LIN {X 0,Y 362.336,Z 282.722,A -85,B 0,C 180,E1 -13021.628,E2 -13021.628} C_VEL
LIN {X 0,Y 361.775,Z 288.928,A -85,B 0,C 180,E1 -13025.313,E2 -13025.313} C_VEL
LIN {X 0,Y 361.344,Z 295.244,A -85,B 0,C 180,E1 -13028.961,E2 -13028.961} C_VEL
LIN {X 0,Y 364.854,Z 309.649,A -85,B 0,C 180,E1 -13029.76,E2 -13029.76} C_VEL
LIN {X 0,Y 366.937,Z 321.069,A -85,B 0,C 180,E1 -13030.541,E2 -13030.541} C_VEL
LIN {X 0,Y 367.97,Z 331.151,A -85,B 0,C 180,E1 -13031.343,E2 -13031.343} C_VEL
LIN {X 0,Y 367.387,Z 339.33,A -85,B 0,C 180,E1 -13032.034,E2 -13032.034} C_VEL
LIN {X 0,Y 366.088,Z 350.021,A -85,B 0,C 180,E1 -13033.121,E2 -13033.121} C_VEL
LIN {X 0,Y 364.817,Z 359.766,A -85,B 0,C 180,E1 -13034.354,E2 -13034.354} C_VEL
LIN {X 0,Y 363.818,Z 368.646,A -85,B 0,C 180,E1 -13035.742,E2 -13035.742} C_VEL
LIN {X 0,Y 362.605,Z 377.356,A -85,B 0,C 180,E1 -13037.406,E2 -13037.406} C_VEL
LIN {X 0,Y 361.765,Z 384.335,A -85,B 0,C 180,E1 -13039.082,E2 -13039.082} C_VEL
LIN {X 0,Y 361.039,Z 390.749,A -85,B 0,C 180,E1 -13041.041,E2 -13041.041} C_VEL
LIN {X 0,Y 360.62,Z 394.992,A -85,B 0,C 180,E1 -13042.723,E2 -13042.723} C_VEL
LIN {X 0,Y 360.393,Z 398.186,A -85,B 0,C 180,E1 -13044.405,E2 -13044.405} C_VEL
LIN {X 0,Y 360.351,Z 399.786,A -85,B 0,C 180,E1 -13045.526,E2 -13045.526} C_VEL
LIN {X 0,Y 360.298,Z 400.979,A -85,B 0,C 180,E1 -13046.645,E2 -13046.645} C_VEL
LIN {X 0,Y 360.304,Z 402.103,A -85,B 0,C 180,E1 -13048.882,E2 -13048.882} C_VEL
LIN {X 0,Y 360.361,Z 402.087,A -85,B 0,C 180,E1 -13050,E2 -13050} C_VEL
LIN {X 0,Y 360.322,Z 401.681,A -85,B 0,C 180,E1 -13051.118,E2 -13051.118} C_VEL
LIN {X 0,Y 360.28,Z 400.838,A -85,B 0,C 180,E1 -13052.236,E2 -13052.236} C_VEL
LIN {X 0,Y 360.304,Z 399.588,A -85,B 0,C 180,E1 -13053.355,E2 -13053.355} C_VEL
LIN {X 0,Y 360.352,Z 396.925,A -85,B 0,C 180,E1 -13055.035,E2 -13055.035} C_VEL
LIN {X 0,Y 360.501,Z 393.232,A -85,B 0,C 180,E1 -13056.717,E2 -13056.717} C_VEL
LIN {X 0,Y 360.762,Z 388.407,A -85,B 0,C 180,E1 -13058.401,E2 -13058.401} C_VEL
LIN {X 0,Y 361.209,Z 382.305,A -85,B 0,C 180,E1 -13060.085,E2 -13060.085} C_VEL
LIN {X 0,Y 361.826,Z 374.701,A -85,B 0,C 180,E1 -13061.768,E2 -13061.768} C_VEL
LIN {X 0,Y 362.586,Z 366.931,A -85,B 0,C 180,E1 -13063.164,E2 -13063.164} C_VEL
LIN {X 0,Y 363.483,Z 356.737,A -85,B 0,C 180,E1 -13064.649,E2 -13064.649} C_VEL
LIN {X 0,Y 364.366,Z 345.554,A -85,B 0,C 180,E1 -13065.953,E2 -13065.953} C_VEL
LIN {X 0,Y 365.33,Z 335.115,A -85,B 0,C 180,E1 -13066.915,E2 -13066.915} C_VEL
LIN {X 0,Y 365.595,Z 328.765,A -85,B 0,C 180,E1 -13067.407,E2 -13067.407} C_VEL
LIN {X 0,Y 364.08,Z 316.069,A -85,B 0,C 180,E1 -13068.276,E2 -13068.276} C_VEL
LIN {X 0,Y 362.102,Z 302.88,A -85,B 0,C 180,E1 -13068.953,E2 -13068.953} C_VEL
LIN {X 0,Y 360.91,Z 295.618,A -85,B 0,C 180,E1 -13069.237,E2 -13069.237} C_VEL
LIN {X 0,Y 361.268,Z 288.936,A -85,B 0,C 180,E1 -13072.896,E2 -13072.896} C_VEL
LIN {X 0,Y 361.707,Z 282.405,A -85,B 0,C 180,E1 -13076.544,E2 -13076.544} C_VEL
LIN {X 0,Y 362.26,Z 275.818,A -85,B 0,C 180,E1 -13080.291,E2 -13080.291} C_VEL
LIN {X 0,Y 362.767,Z 270.224,A -85,B 0,C 180,E1 -13083.585,E2 -13083.585} C_VEL
LIN {X 0,Y 363.011,Z 265.914,A -85,B 0,C 180,E1 -13086.19,E2 -13086.19} C_VEL
LIN {X 0,Y 362.596,Z 262.575,A -85,B 0,C 180,E1 -13088.333,E2 -13088.333} C_VEL
LIN {X 0,Y 361.875,Z 258.411,A -85,B 0,C 180,E1 -13091.166,E2 -13091.166} C_VEL
LIN {X 0,Y 361.803,Z 258.415,A -85,B 0,C 180,E1 -13094.369,E2 -13094.369} C_VEL
LIN {X 0,Y 361.811,Z 258.414,A -85,B 0,C 180,E1 -13097.571,E2 -13097.571} C_VEL
LIN {X 0,Y 361.839,Z 258.41,A -85,B 0,C 180,E1 -13101.57,E2 -13101.57} C_VEL
LIN {X 0,Y 361.867,Z 258.412,A -85,B 0,C 180,E1 -13104.655,E2 -13104.655} C_VEL
LIN {X 0,Y 361.835,Z 258.414,A -85,B 0,C 180,E1 -13108.369,E2 -13108.369} C_VEL
LIN {X 0,Y 361.863,Z 258.41,A -85,B 0,C 180,E1 -13110.951,E2 -13110.951} C_VEL
LIN {X 0,Y 361.878,Z 258.409,A -85,B 0,C 180,E1 -13114.705,E2 -13114.705} C_VEL
LIN {X 0,Y 361.85,Z 258.414,A -85,B 0,C 180,E1 -13118.343,E2 -13118.343} C_VEL
LIN {X 0,Y 361.963,Z 258.398,A -85,B 0,C 180,E1 -13122.06,E2 -13122.06} C_VEL
LIN {X 0,Y 361.992,Z 258.396,A -85,B 0,C 180,E1 -13126.1,E2 -13126.1} C_VEL
LIN {X 0,Y 362.025,Z 258.391,A -85,B 0,C 180,E1 -13129.937,E2 -13129.937} C_VEL
LIN {X 0,Y 362.155,Z 258.371,A -85,B 0,C 180,E1 -13133.312,E2 -13133.312} C_VEL
LIN {X 0,Y 362.274,Z 258.361,A -85,B 0,C 180,E1 -13137.775,E2 -13137.775} C_VEL
LIN {X 0,Y 362.421,Z 258.343,A -85,B 0,C 180,E1 -13139.999,E2 -13139.999} C_VEL
LIN {X 0,Y 362.275,Z 258.358,A -85,B 0,C 180,E1 -13142.222,E2 -13142.222} C_VEL
LIN {X 0,Y 362.164,Z 258.37,A -85,B 0,C 180,E1 -13146.685,E2 -13146.685} C_VEL
LIN {X 0,Y 362.065,Z 258.382,A -85,B 0,C 180,E1 -13148.932,E2 -13148.932} C_VEL
LIN {X 0,Y 361.951,Z 258.397,A -85,B 0,C 180,E1 -13152.331,E2 -13152.331} C_VEL
LIN {X 0,Y 361.952,Z 258.396,A -85,B 0,C 180,E1 -13154.619,E2 -13154.619} C_VEL
LIN {X 0,Y 361.946,Z 258.398,A -85,B 0,C 180,E1 -13158.098,E2 -13158.098} C_VEL
LIN {X 0,Y 361.882,Z 258.408,A -85,B 0,C 180,E1 -13161.652,E2 -13161.652} C_VEL
LIN {X 0,Y 361.918,Z 258.405,A -85,B 0,C 180,E1 -13165.289,E2 -13165.289} C_VEL
LIN {X 0,Y 361.912,Z 258.402,A -85,B 0,C 180,E1 -13167.777,E2 -13167.777} C_VEL
LIN {X 0,Y 361.836,Z 258.415,A -85,B 0,C 180,E1 -13171.284,E2 -13171.284} C_VEL
LIN {X 0,Y 361.843,Z 258.409,A -85,B 0,C 180,E1 -13174.28,E2 -13174.28} C_VEL
LIN {X 0,Y 361.854,Z 258.412,A -85,B 0,C 180,E1 -13177.223,E2 -13177.223} C_VEL
LIN {X 0,Y 361.894,Z 258.407,A -85,B 0,C 180,E1 -13180.768,E2 -13180.768} C_VEL
LIN {X 0,Y 361.892,Z 258.404,A -85,B 0,C 180,E1 -13184.354,E2 -13184.354} C_VEL
LIN {X 0,Y 361.826,Z 258.411,A -85,B 0,C 180,E1 -13187.567,E2 -13187.567} C_VEL
LIN {X 0,Y 361.86,Z 258.407,A -85,B 0,C 180,E1 -13191.575,E2 -13191.575} C_VEL
LIN {X 0,Y 361.863,Z 258.412,A -85,B 0,C 180,E1 -13194.655,E2 -13194.655} C_VEL
LIN {X 0,Y 361.826,Z 258.416,A -85,B 0,C 180,E1 -13198.37,E2 -13198.37} C_VEL
LIN {X 0,Y 361.889,Z 258.405,A -85,B 0,C 180,E1 -13200.955,E2 -13200.955} C_VEL
LIN {X 0,Y 361.904,Z 258.402,A -85,B 0,C 180,E1 -13203.472,E2 -13203.472} C_VEL
LIN {X 0,Y 361.737,Z 258.423,A -85,B 0,C 180,E1 -13207.135,E2 -13207.135} C_VEL
LIN {X 0,Y 361.647,Z 258.533,A -85,B 0,C 180,E1 -13208.332,E2 -13208.332} C_VEL
LIN {X 0,Y 361.516,Z 262.687,A -85,B 0,C 180,E1 -13211.878,E2 -13211.878} C_VEL
LIN {X 0,Y 361.312,Z 266.846,A -85,B 0,C 180,E1 -13215.353,E2 -13215.353} C_VEL
LIN {X 0,Y 361.258,Z 269.647,A -85,B 0,C 180,E1 -13217.644,E2 -13217.644} C_VEL
LIN {X 0,Y 361.091,Z 275.315,A -85,B 0,C 180,E1 -13222.17,E2 -13222.17} C_VEL
LIN {X 0,Y 361.062,Z 277.456,A -85,B 0,C 180,E1 -13223.854,E2 -13223.854} C_VEL
LIN {X 0,Y 364.211,Z 293.091,A -85,B 0,C 180,E1 -13224.62,E2 -13224.62} C_VEL
LIN {X 0,Y 365.873,Z 303.958,A -85,B 0,C 180,E1 -13225.317,E2 -13225.317} C_VEL
LIN {X 0,Y 366.247,Z 307.745,A -85,B 0,C 180,E1 -13225.598,E2 -13225.598} C_VEL
LIN {X 0,Y 365.413,Z 319.726,A -85,B 0,C 180,E1 -13226.554,E2 -13226.554} C_VEL
LIN {X 0,Y 364.435,Z 330.442,A -85,B 0,C 180,E1 -13227.651,E2 -13227.651} C_VEL
LIN {X 0,Y 363.634,Z 340.162,A -85,B 0,C 180,E1 -13228.893,E2 -13228.893} C_VEL
LIN {X 0,Y 362.785,Z 349.037,A -85,B 0,C 180,E1 -13230.277,E2 -13230.277} C_VEL
LIN {X 0,Y 361.891,Z 357.719,A -85,B 0,C 180,E1 -13231.947,E2 -13231.947} C_VEL
LIN {X 0,Y 361.339,Z 364.629,A -85,B 0,C 180,E1 -13233.624,E2 -13233.624} C_VEL
LIN {X 0,Y 360.896,Z 370.979,A -85,B 0,C 180,E1 -13235.587,E2 -13235.587} C_VEL
LIN {X 0,Y 360.605,Z 375.157,A -85,B 0,C 180,E1 -13237.278,E2 -13237.278} C_VEL
LIN {X 0,Y 360.348,Z 378.28,A -85,B 0,C 180,E1 -13238.976,E2 -13238.976} C_VEL
LIN {X 0,Y 360.217,Z 379.833,A -85,B 0,C 180,E1 -13240.113,E2 -13240.113} C_VEL
LIN {X 0,Y 360.222,Z 380.918,A -85,B 0,C 180,E1 -13241.25,E2 -13241.25} C_VEL
LIN {X 0,Y 360.241,Z 381.748,A -85,B 0,C 180,E1 -13242.728,E2 -13242.728} C_VEL
LIN {X 0,Y 360.186,Z 381.776,A -85,B 0,C 180,E1 -13244.694,E2 -13244.694} C_VEL
LIN {X 0,Y 360.264,Z 381.203,A -85,B 0,C 180,E1 -13245.849,E2 -13245.849} C_VEL
LIN {X 0,Y 360.421,Z 380.065,A -85,B 0,C 180,E1 -13247.169,E2 -13247.169} C_VEL
LIN {X 0,Y 360.538,Z 378.83,A -85,B 0,C 180,E1 -13248.173,E2 -13248.173} C_VEL
LIN {X 0,Y 360.934,Z 375.84,A -85,B 0,C 180,E1 -13249.922,E2 -13249.922} C_VEL
LIN {X 0,Y 361.452,Z 371.724,A -85,B 0,C 180,E1 -13251.68,E2 -13251.68} C_VEL
LIN {X 0,Y 362.307,Z 365.284,A -85,B 0,C 180,E1 -13253.734,E2 -13253.734} C_VEL
LIN {X 0,Y 363.259,Z 358.194,A -85,B 0,C 180,E1 -13255.497,E2 -13255.497} C_VEL
LIN {X 0,Y 364.281,Z 350.879,A -85,B 0,C 180,E1 -13256.96,E2 -13256.96} C_VEL
LIN {X 0,Y 365.571,Z 340.89,A -85,B 0,C 180,E1 -13258.568,E2 -13258.568} C_VEL
LIN {X 0,Y 366.821,Z 330.741,A -85,B 0,C 180,E1 -13259.876,E2 -13259.876} C_VEL
LIN {X 0,Y 368.047,Z 319.433,A -85,B 0,C 180,E1 -13261.035,E2 -13261.035} C_VEL
LIN {X 0,Y 369.002,Z 309.168,A -85,B 0,C 180,E1 -13261.865,E2 -13261.865} C_VEL
LIN {X 0,Y 366.904,Z 298.129,A -85,B 0,C 180,E1 -13262.76,E2 -13262.76} C_VEL
LIN {X 0,Y 363.301,Z 285.154,A -85,B 0,C 180,E1 -13263.657,E2 -13263.657} C_VEL
LIN {X 0,Y 361.812,Z 280.58,A -85,B 0,C 180,E1 -13263.932,E2 -13263.932} C_VEL
LIN {X 0,Y 360.522,Z 278.624,A -85,B 0,C 180,E1 -13264.212,E2 -13264.212} C_VEL
LIN {X 0,Y 358.666,Z 277.299,A -85,B 0,C 180,E1 -13264.811,E2 -13264.811} C_VEL
LIN {X 0,Y 356.413,Z 276.288,A -85,B 0,C 180,E1 -13265.902,E2 -13265.902} C_VEL
LIN {X 0,Y 354.793,Z 275.058,A -85,B 0,C 180,E1 -13267.289,E2 -13267.289} C_VEL
LIN {X 0,Y 354.295,Z 273.377,A -85,B 0,C 180,E1 -13268.691,E2 -13268.691} C_VEL
LIN {X 0,Y 354.635,Z 269.309,A -85,B 0,C 180,E1 -13272.359,E2 -13272.359} C_VEL
LIN {X 0,Y 354.935,Z 265.981,A -85,B 0,C 180,E1 -13275.464,E2 -13275.464} C_VEL
LIN {X 0,Y 355.072,Z 262.602,A -85,B 0,C 180,E1 -13278.774,E2 -13278.774} C_VEL
LIN {X 0,Y 354.969,Z 260.745,A -85,B 0,C 180,E1 -13280.689,E2 -13280.689} C_VEL
LIN {X 0,Y 354.802,Z 259.292,A -85,B 0,C 180,E1 -13282.402,E2 -13282.402} C_VEL
LIN {X 0,Y 354.8,Z 259.293,A -85,B 0,C 180,E1 -13284.942,E2 -13284.942} C_VEL
LIN {X 0,Y 354.782,Z 259.295,A -85,B 0,C 180,E1 -13288.406,E2 -13288.406} C_VEL
LIN {X 0,Y 354.842,Z 259.285,A -85,B 0,C 180,E1 -13291.62,E2 -13291.62} C_VEL
LIN {X 0,Y 354.889,Z 259.279,A -85,B 0,C 180,E1 -13294.174,E2 -13294.174} C_VEL
LIN {X 0,Y 354.843,Z 259.286,A -85,B 0,C 180,E1 -13297.896,E2 -13297.896} C_VEL
LIN {X 0,Y 354.913,Z 259.275,A -85,B 0,C 180,E1 -13301.892,E2 -13301.892} C_VEL
LIN {X 0,Y 354.933,Z 259.271,A -85,B 0,C 180,E1 -13305.982,E2 -13305.982} C_VEL
LIN {X 0,Y 354.968,Z 259.27,A -85,B 0,C 180,E1 -13309.737,E2 -13309.737} C_VEL
LIN {X 0,Y 355.116,Z 259.25,A -85,B 0,C 180,E1 -13313.182,E2 -13313.182} C_VEL
LIN {X 0,Y 355.238,Z 259.236,A -85,B 0,C 180,E1 -13317.734,E2 -13317.734} C_VEL
LIN {X 0,Y 355.365,Z 259.218,A -85,B 0,C 180,E1 -13320.001,E2 -13320.001} C_VEL
LIN {X 0,Y 355.237,Z 259.237,A -85,B 0,C 180,E1 -13322.269,E2 -13322.269} C_VEL
LIN {X 0,Y 355.129,Z 259.25,A -85,B 0,C 180,E1 -13326.821,E2 -13326.821} C_VEL
LIN {X 0,Y 355.008,Z 259.265,A -85,B 0,C 180,E1 -13329.114,E2 -13329.114} C_VEL
LIN {X 0,Y 354.915,Z 259.279,A -85,B 0,C 180,E1 -13332.582,E2 -13332.582} C_VEL
LIN {X 0,Y 354.883,Z 259.282,A -85,B 0,C 180,E1 -13336.097,E2 -13336.097} C_VEL
LIN {X 0,Y 354.901,Z 259.283,A -85,B 0,C 180,E1 -13338.473,E2 -13338.473} C_VEL
LIN {X 0,Y 354.83,Z 259.291,A -85,B 0,C 180,E1 -13342.108,E2 -13342.108} C_VEL
LIN {X 0,Y 354.869,Z 259.288,A -85,B 0,C 180,E1 -13345.831,E2 -13345.831} C_VEL
